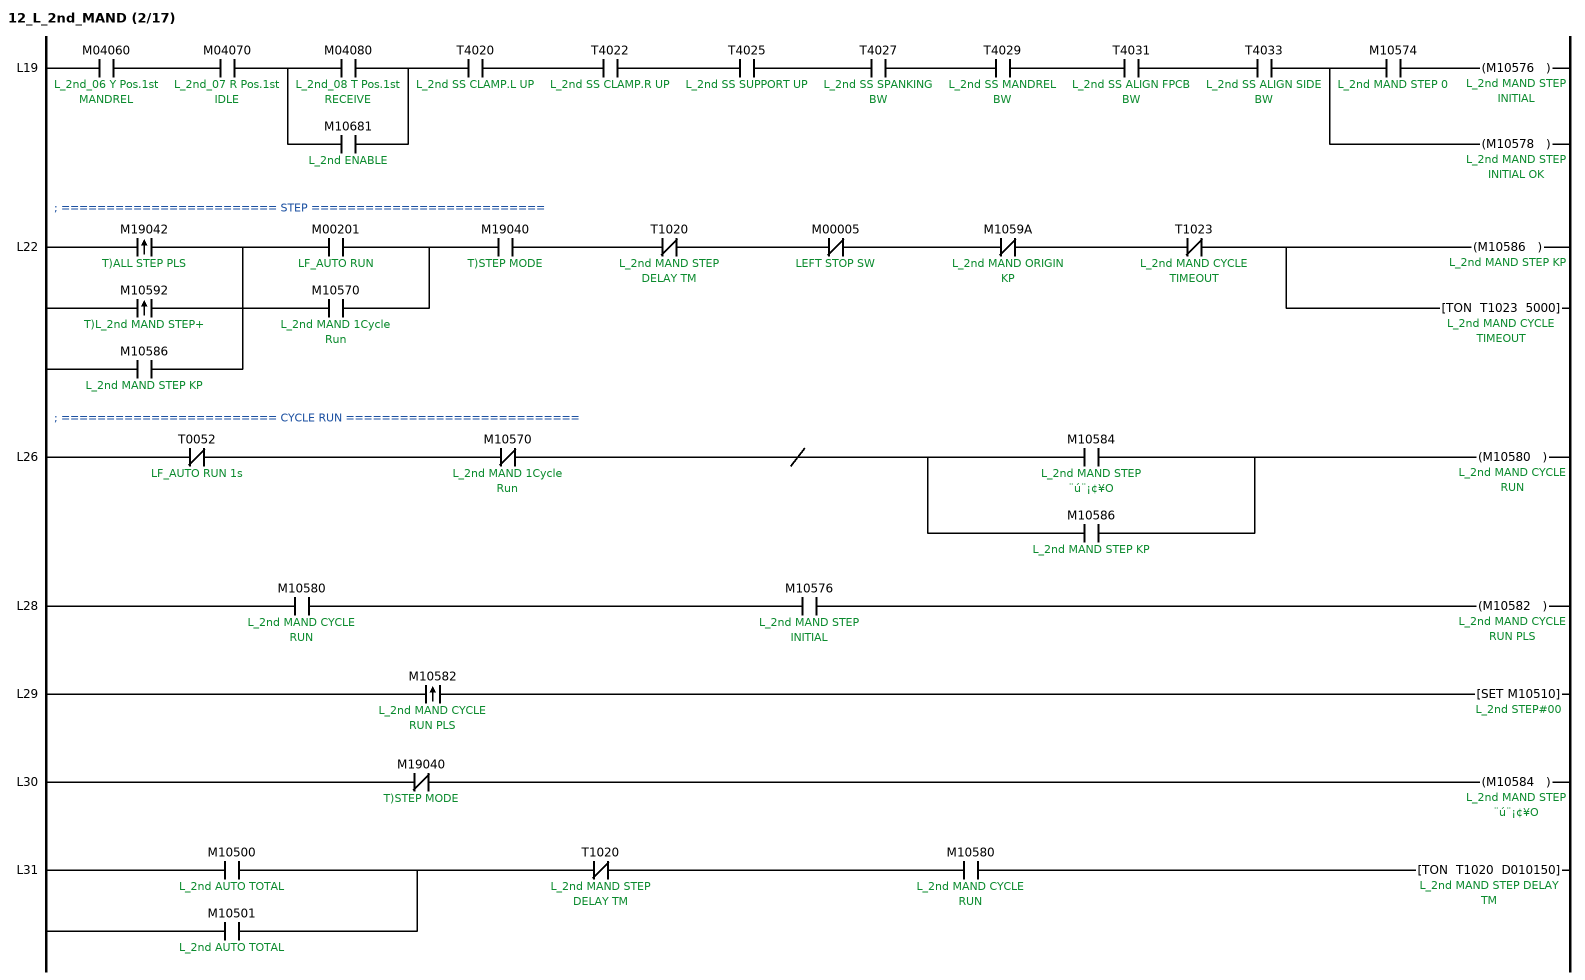
[picture p72: 12_L_2nd_MAND rungs L19-L31]
; L19
LOAD      M04060	// L_2nd_06 Y Pos.1st MANDREL
AND       M04070	// L_2nd_07 R Pos.1st IDLE
LOAD      M04080	// L_2nd_08 T Pos.1st RECEIVE
OR        M10681	// L_2nd ENABLE
AND LOAD
AND       T4020	// L_2nd SS CLAMP.L UP
AND       T4022	// L_2nd SS CLAMP.R UP
AND       T4025	// L_2nd SS SUPPORT UP
AND       T4027	// L_2nd SS SPANKING BW
AND       T4029	// L_2nd SS MANDREL BW
AND       T4031	// L_2nd SS ALIGN FPCB BW
AND       T4033	// L_2nd SS ALIGN SIDE BW
MPUSH
AND       M10574	// L_2nd MAND STEP 0
OUT       M10576	// L_2nd MAND STEP INITIAL
MPOP
OUT       M10578	// L_2nd MAND STEP INITIAL OK
// ======================== STEP ==========================
; L22
LOADP     M19042	// T)ALL STEP PLS
ORP       M10592	// T)L_2nd MAND STEP+
OR        M10586	// L_2nd MAND STEP KP
LOAD      M00201	// LF_AUTO RUN
OR        M10570	// L_2nd MAND 1Cycle Run
AND LOAD
AND       M19040	// T)STEP MODE
AND NOT   T1020	// L_2nd MAND STEP DELAY TM
AND NOT   M00005	// LEFT STOP SW
AND NOT   M1059A	// L_2nd MAND ORIGIN KP
AND NOT   T1023	// L_2nd MAND CYCLE TIMEOUT
OUT       M10586	// L_2nd MAND STEP KP
TON       T1023 5000	// L_2nd MAND CYCLE TIMEOUT
// ======================== CYCLE RUN ==========================
; L26
LOAD NOT  T0052	// LF_AUTO RUN 1s
AND NOT   M10570	// L_2nd MAND 1Cycle Run
NOT
LOAD      M10584	// L_2nd MAND STEP ¨ú¨¡¢¥O
OR        M10586	// L_2nd MAND STEP KP
AND LOAD
OUT       M10580	// L_2nd MAND CYCLE RUN
; L28
LOAD      M10580	// L_2nd MAND CYCLE RUN
AND       M10576	// L_2nd MAND STEP INITIAL
OUT       M10582	// L_2nd MAND CYCLE RUN PLS
; L29
LOADP     M10582	// L_2nd MAND CYCLE RUN PLS
SET       M10510	// L_2nd STEP#00
; L30
LOAD NOT  M19040	// T)STEP MODE
OUT       M10584	// L_2nd MAND STEP ¨ú¨¡¢¥O
; L31
LOAD      M10500	// L_2nd AUTO TOTAL
OR        M10501	// L_2nd AUTO TOTAL
AND NOT   T1020	// L_2nd MAND STEP DELAY TM
AND       M10580	// L_2nd MAND CYCLE RUN
TON       T1020 D010150	// L_2nd MAND STEP DELAY TM

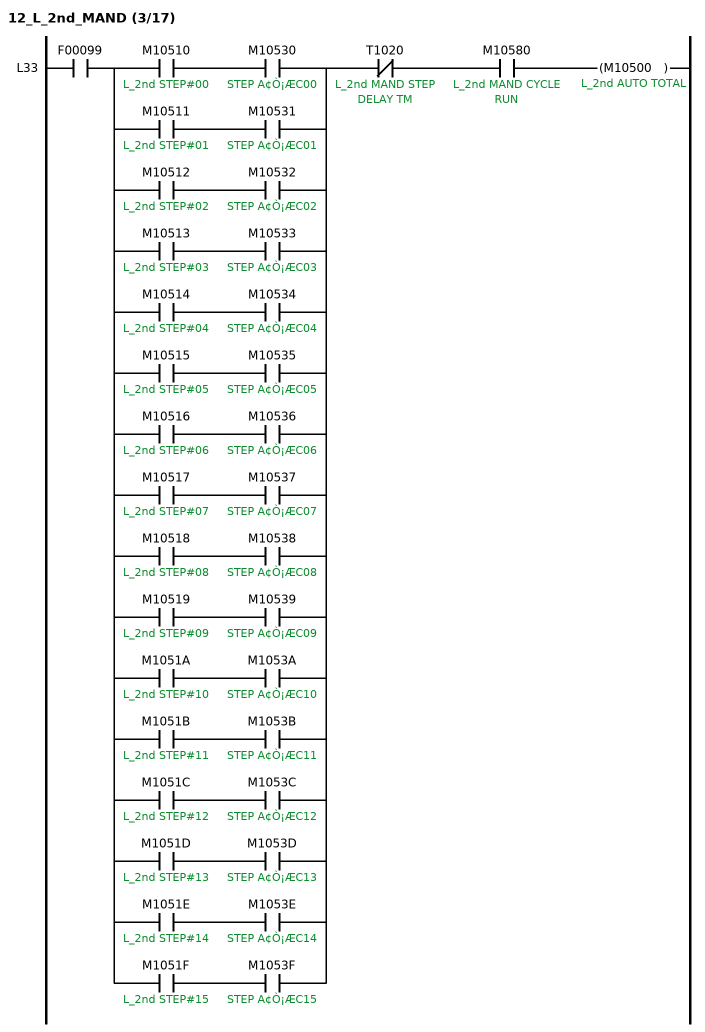
; L33
LOAD      F00099
LOAD      M10510	// L_2nd STEP#00
AND       M10530	// STEP A¢Ò¡ÆC00
LOAD      M10511	// L_2nd STEP#01
AND       M10531	// STEP A¢Ò¡ÆC01
OR LOAD
LOAD      M10512	// L_2nd STEP#02
AND       M10532	// STEP A¢Ò¡ÆC02
OR LOAD
LOAD      M10513	// L_2nd STEP#03
AND       M10533	// STEP A¢Ò¡ÆC03
OR LOAD
LOAD      M10514	// L_2nd STEP#04
AND       M10534	// STEP A¢Ò¡ÆC04
OR LOAD
LOAD      M10515	// L_2nd STEP#05
AND       M10535	// STEP A¢Ò¡ÆC05
OR LOAD
LOAD      M10516	// L_2nd STEP#06
AND       M10536	// STEP A¢Ò¡ÆC06
OR LOAD
LOAD      M10517	// L_2nd STEP#07
AND       M10537	// STEP A¢Ò¡ÆC07
OR LOAD
LOAD      M10518	// L_2nd STEP#08
AND       M10538	// STEP A¢Ò¡ÆC08
OR LOAD
LOAD      M10519	// L_2nd STEP#09
AND       M10539	// STEP A¢Ò¡ÆC09
OR LOAD
LOAD      M1051A	// L_2nd STEP#10
AND       M1053A	// STEP A¢Ò¡ÆC10
OR LOAD
LOAD      M1051B	// L_2nd STEP#11
AND       M1053B	// STEP A¢Ò¡ÆC11
OR LOAD
LOAD      M1051C	// L_2nd STEP#12
AND       M1053C	// STEP A¢Ò¡ÆC12
OR LOAD
LOAD      M1051D	// L_2nd STEP#13
AND       M1053D	// STEP A¢Ò¡ÆC13
OR LOAD
LOAD      M1051E	// L_2nd STEP#14
AND       M1053E	// STEP A¢Ò¡ÆC14
OR LOAD
LOAD      M1051F	// L_2nd STEP#15
AND       M1053F	// STEP A¢Ò¡ÆC15
OR LOAD
AND LOAD
AND NOT   T1020	// L_2nd MAND STEP DELAY TM
AND       M10580	// L_2nd MAND CYCLE RUN
OUT       M10500	// L_2nd AUTO TOTAL

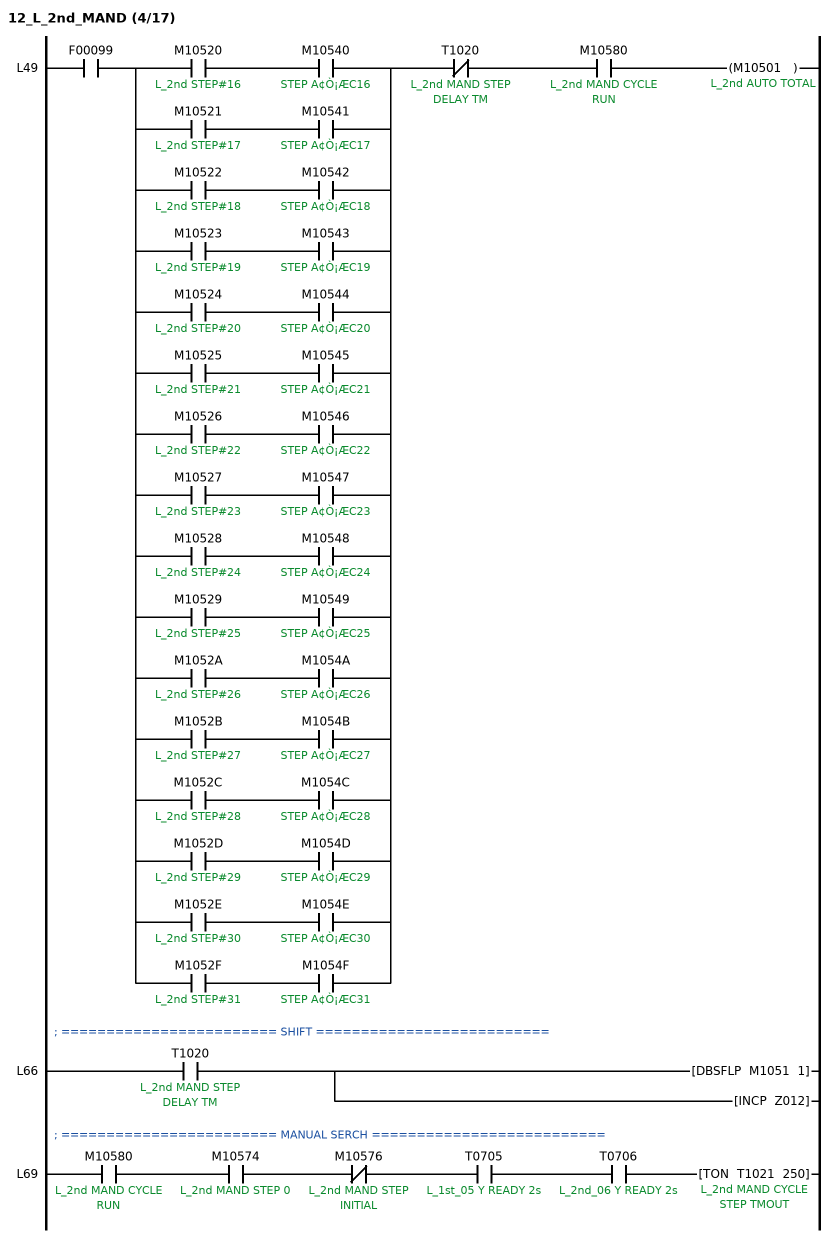
; L49
LOAD      F00099
LOAD      M10520	// L_2nd STEP#16
AND       M10540	// STEP A¢Ò¡ÆC16
LOAD      M10521	// L_2nd STEP#17
AND       M10541	// STEP A¢Ò¡ÆC17
OR LOAD
LOAD      M10522	// L_2nd STEP#18
AND       M10542	// STEP A¢Ò¡ÆC18
OR LOAD
LOAD      M10523	// L_2nd STEP#19
AND       M10543	// STEP A¢Ò¡ÆC19
OR LOAD
LOAD      M10524	// L_2nd STEP#20
AND       M10544	// STEP A¢Ò¡ÆC20
OR LOAD
LOAD      M10525	// L_2nd STEP#21
AND       M10545	// STEP A¢Ò¡ÆC21
OR LOAD
LOAD      M10526	// L_2nd STEP#22
AND       M10546	// STEP A¢Ò¡ÆC22
OR LOAD
LOAD      M10527	// L_2nd STEP#23
AND       M10547	// STEP A¢Ò¡ÆC23
OR LOAD
LOAD      M10528	// L_2nd STEP#24
AND       M10548	// STEP A¢Ò¡ÆC24
OR LOAD
LOAD      M10529	// L_2nd STEP#25
AND       M10549	// STEP A¢Ò¡ÆC25
OR LOAD
LOAD      M1052A	// L_2nd STEP#26
AND       M1054A	// STEP A¢Ò¡ÆC26
OR LOAD
LOAD      M1052B	// L_2nd STEP#27
AND       M1054B	// STEP A¢Ò¡ÆC27
OR LOAD
LOAD      M1052C	// L_2nd STEP#28
AND       M1054C	// STEP A¢Ò¡ÆC28
OR LOAD
LOAD      M1052D	// L_2nd STEP#29
AND       M1054D	// STEP A¢Ò¡ÆC29
OR LOAD
LOAD      M1052E	// L_2nd STEP#30
AND       M1054E	// STEP A¢Ò¡ÆC30
OR LOAD
LOAD      M1052F	// L_2nd STEP#31
AND       M1054F	// STEP A¢Ò¡ÆC31
OR LOAD
AND LOAD
AND NOT   T1020	// L_2nd MAND STEP DELAY TM
AND       M10580	// L_2nd MAND CYCLE RUN
OUT       M10501	// L_2nd AUTO TOTAL
// ======================== SHIFT ==========================
; L66
LOAD      T1020	// L_2nd MAND STEP DELAY TM
DBSFLP    M1051 1
INCP      Z012
// ======================== MANUAL SERCH ==========================
; L69
LOAD      M10580	// L_2nd MAND CYCLE RUN
AND       M10574	// L_2nd MAND STEP 0
AND NOT   M10576	// L_2nd MAND STEP INITIAL
AND       T0705	// L_1st_05 Y READY 2s
AND       T0706	// L_2nd_06 Y READY 2s
TON       T1021 250	// L_2nd MAND CYCLE STEP TMOUT

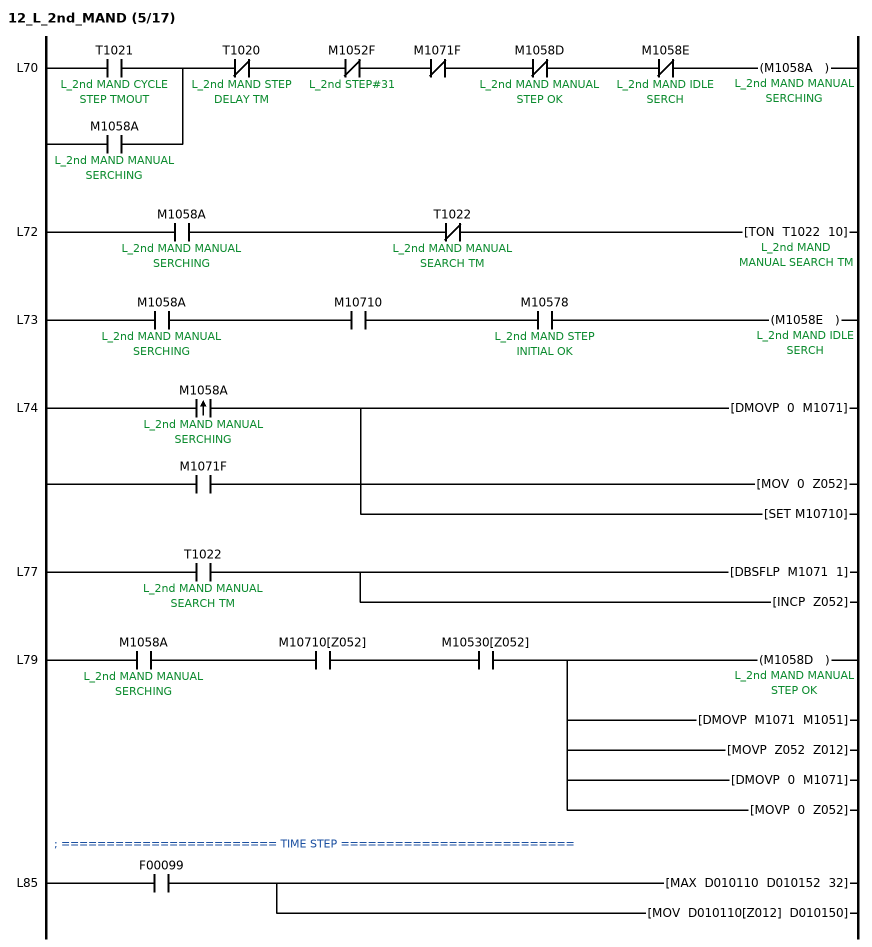
; L70
LOAD      T1021	// L_2nd MAND CYCLE STEP TMOUT
OR        M1058A	// L_2nd MAND MANUAL SERCHING
AND NOT   T1020	// L_2nd MAND STEP DELAY TM
AND NOT   M1052F	// L_2nd STEP#31
AND NOT   M1071F
AND NOT   M1058D	// L_2nd MAND MANUAL STEP OK
AND NOT   M1058E	// L_2nd MAND IDLE SERCH
OUT       M1058A	// L_2nd MAND MANUAL SERCHING
; L72
LOAD      M1058A	// L_2nd MAND MANUAL SERCHING
AND NOT   T1022	// L_2nd MAND MANUAL SEARCH TM
TON       T1022 10	// L_2nd MAND MANUAL SEARCH TM
; L73
LOAD      M1058A	// L_2nd MAND MANUAL SERCHING
AND       M10710
AND       M10578	// L_2nd MAND STEP INITIAL OK
OUT       M1058E	// L_2nd MAND IDLE SERCH
; L74
LOADP     M1058A	// L_2nd MAND MANUAL SERCHING
OR        M1071F
DMOVP     0 M1071
MOV       0 Z052
SET       M10710
; L77
LOAD      T1022	// L_2nd MAND MANUAL SEARCH TM
DBSFLP    M1071 1
INCP      Z052
; L79
LOAD      M1058A	// L_2nd MAND MANUAL SERCHING
AND       M10710[Z052]
AND       M10530[Z052]
OUT       M1058D	// L_2nd MAND MANUAL STEP OK
DMOVP     M1071 M1051
MOVP      Z052 Z012
DMOVP     0 M1071
MOVP      0 Z052
// ======================== TIME STEP ==========================
; L85
LOAD      F00099
MAX       D010110 D010152 32
MOV       D010110[Z012] D010150

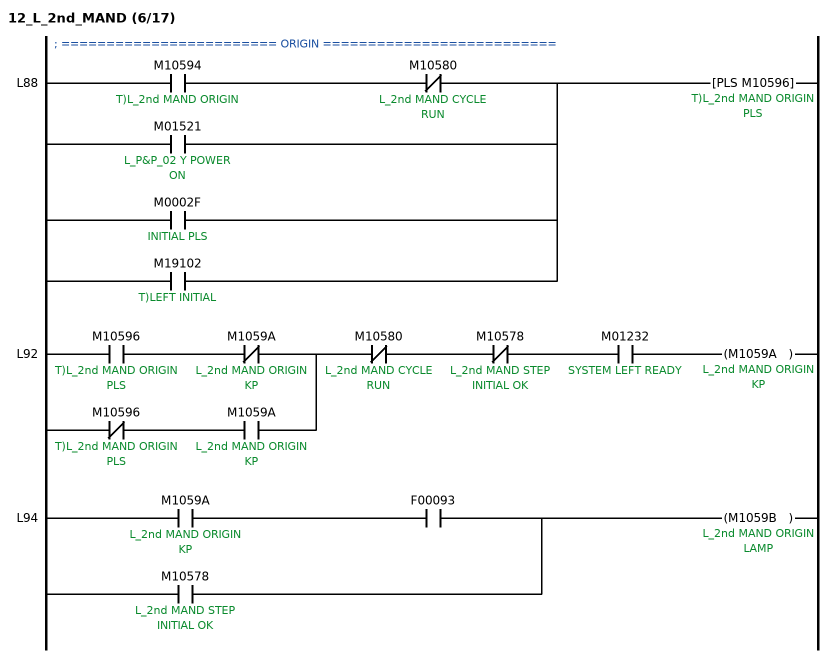
// ======================== ORIGIN ==========================
; L88
LOAD      M10594	// T)L_2nd MAND ORIGIN
AND NOT   M10580	// L_2nd MAND CYCLE RUN
OR        M01521	// L_P&P_02 Y POWER ON
OR        M0002F	// INITIAL PLS
OR        M19102	// T)LEFT INITIAL
OUTP      M10596	// T)L_2nd MAND ORIGIN PLS
; L92
LOAD      M10596	// T)L_2nd MAND ORIGIN PLS
AND NOT   M1059A	// L_2nd MAND ORIGIN KP
LOAD NOT  M10596	// T)L_2nd MAND ORIGIN PLS
AND       M1059A	// L_2nd MAND ORIGIN KP
OR LOAD
AND NOT   M10580	// L_2nd MAND CYCLE RUN
AND NOT   M10578	// L_2nd MAND STEP INITIAL OK
AND       M01232	// SYSTEM LEFT READY
OUT       M1059A	// L_2nd MAND ORIGIN KP
; L94
LOAD      M1059A	// L_2nd MAND ORIGIN KP
AND       F00093
OR        M10578	// L_2nd MAND STEP INITIAL OK
OUT       M1059B	// L_2nd MAND ORIGIN LAMP

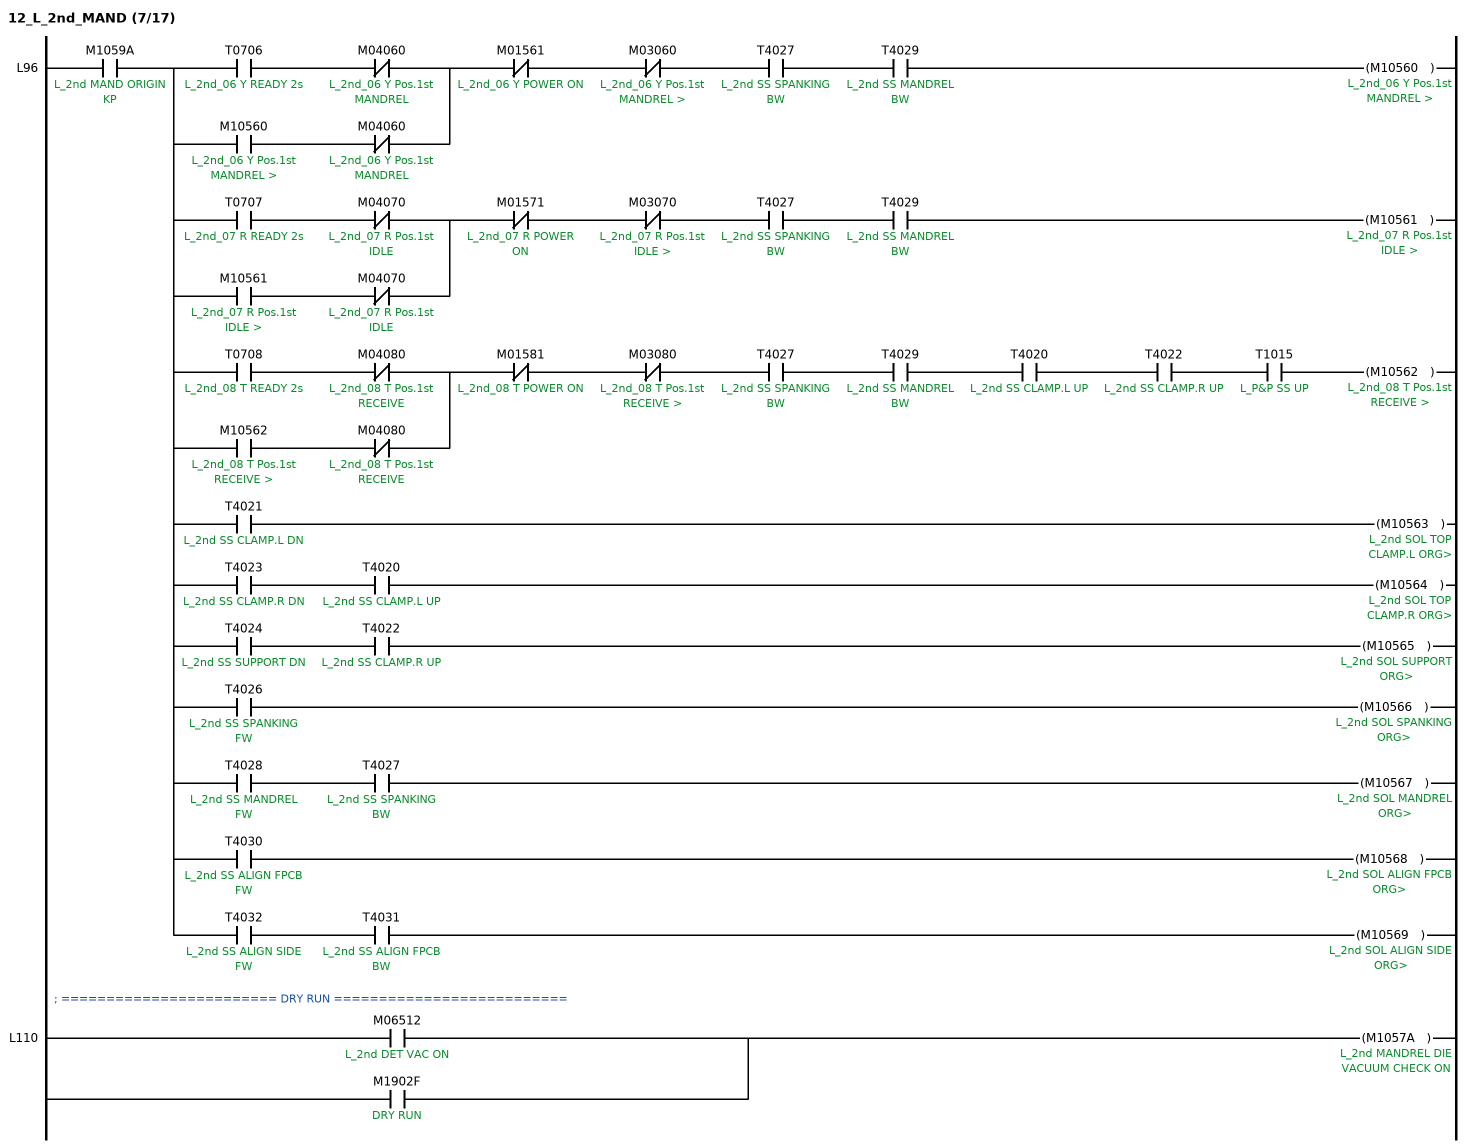
; L96
LOAD      M1059A	// L_2nd MAND ORIGIN KP
MPUSH
LOAD      T0706	// L_2nd_06 Y READY 2s
AND NOT   M04060	// L_2nd_06 Y Pos.1st MANDREL
LOAD      M10560	// L_2nd_06 Y Pos.1st MANDREL >
AND NOT   M04060	// L_2nd_06 Y Pos.1st MANDREL
OR LOAD
AND LOAD
AND NOT   M01561	// L_2nd_06 Y POWER ON
AND NOT   M03060	// L_2nd_06 Y Pos.1st MANDREL >
AND       T4027	// L_2nd SS SPANKING BW
AND       T4029	// L_2nd SS MANDREL BW
OUT       M10560	// L_2nd_06 Y Pos.1st MANDREL >
MLOAD
LOAD      T0707	// L_2nd_07 R READY 2s
AND NOT   M04070	// L_2nd_07 R Pos.1st IDLE
LOAD      M10561	// L_2nd_07 R Pos.1st IDLE >
AND NOT   M04070	// L_2nd_07 R Pos.1st IDLE
OR LOAD
AND LOAD
AND NOT   M01571	// L_2nd_07 R POWER ON
AND NOT   M03070	// L_2nd_07 R Pos.1st IDLE >
AND       T4027	// L_2nd SS SPANKING BW
AND       T4029	// L_2nd SS MANDREL BW
OUT       M10561	// L_2nd_07 R Pos.1st IDLE >
MLOAD
LOAD      T0708	// L_2nd_08 T READY 2s
AND NOT   M04080	// L_2nd_08 T Pos.1st RECEIVE
LOAD      M10562	// L_2nd_08 T Pos.1st RECEIVE >
AND NOT   M04080	// L_2nd_08 T Pos.1st RECEIVE
OR LOAD
AND LOAD
AND NOT   M01581	// L_2nd_08 T POWER ON
AND NOT   M03080	// L_2nd_08 T Pos.1st RECEIVE >
AND       T4027	// L_2nd SS SPANKING BW
AND       T4029	// L_2nd SS MANDREL BW
AND       T4020	// L_2nd SS CLAMP.L UP
AND       T4022	// L_2nd SS CLAMP.R UP
AND       T1015	// L_P&P SS UP
OUT       M10562	// L_2nd_08 T Pos.1st RECEIVE >
MLOAD
AND       T4021	// L_2nd SS CLAMP.L DN
OUT       M10563	// L_2nd SOL TOP CLAMP.L ORG>
MLOAD
AND       T4023	// L_2nd SS CLAMP.R DN
AND       T4020	// L_2nd SS CLAMP.L UP
OUT       M10564	// L_2nd SOL TOP CLAMP.R ORG>
MLOAD
AND       T4024	// L_2nd SS SUPPORT DN
AND       T4022	// L_2nd SS CLAMP.R UP
OUT       M10565	// L_2nd SOL SUPPORT ORG>
MLOAD
AND       T4026	// L_2nd SS SPANKING FW
OUT       M10566	// L_2nd SOL SPANKING ORG>
MLOAD
AND       T4028	// L_2nd SS MANDREL FW
AND       T4027	// L_2nd SS SPANKING BW
OUT       M10567	// L_2nd SOL MANDREL ORG>
MLOAD
AND       T4030	// L_2nd SS ALIGN FPCB FW
OUT       M10568	// L_2nd SOL ALIGN FPCB ORG>
MPOP
AND       T4032	// L_2nd SS ALIGN SIDE FW
AND       T4031	// L_2nd SS ALIGN FPCB BW
OUT       M10569	// L_2nd SOL ALIGN SIDE ORG>
// ======================== DRY RUN ==========================
; L110
LOAD      M06512	// L_2nd DET VAC ON
OR        M1902F	// DRY RUN
OUT       M1057A	// L_2nd MANDREL DIE VACUUM CHECK ON

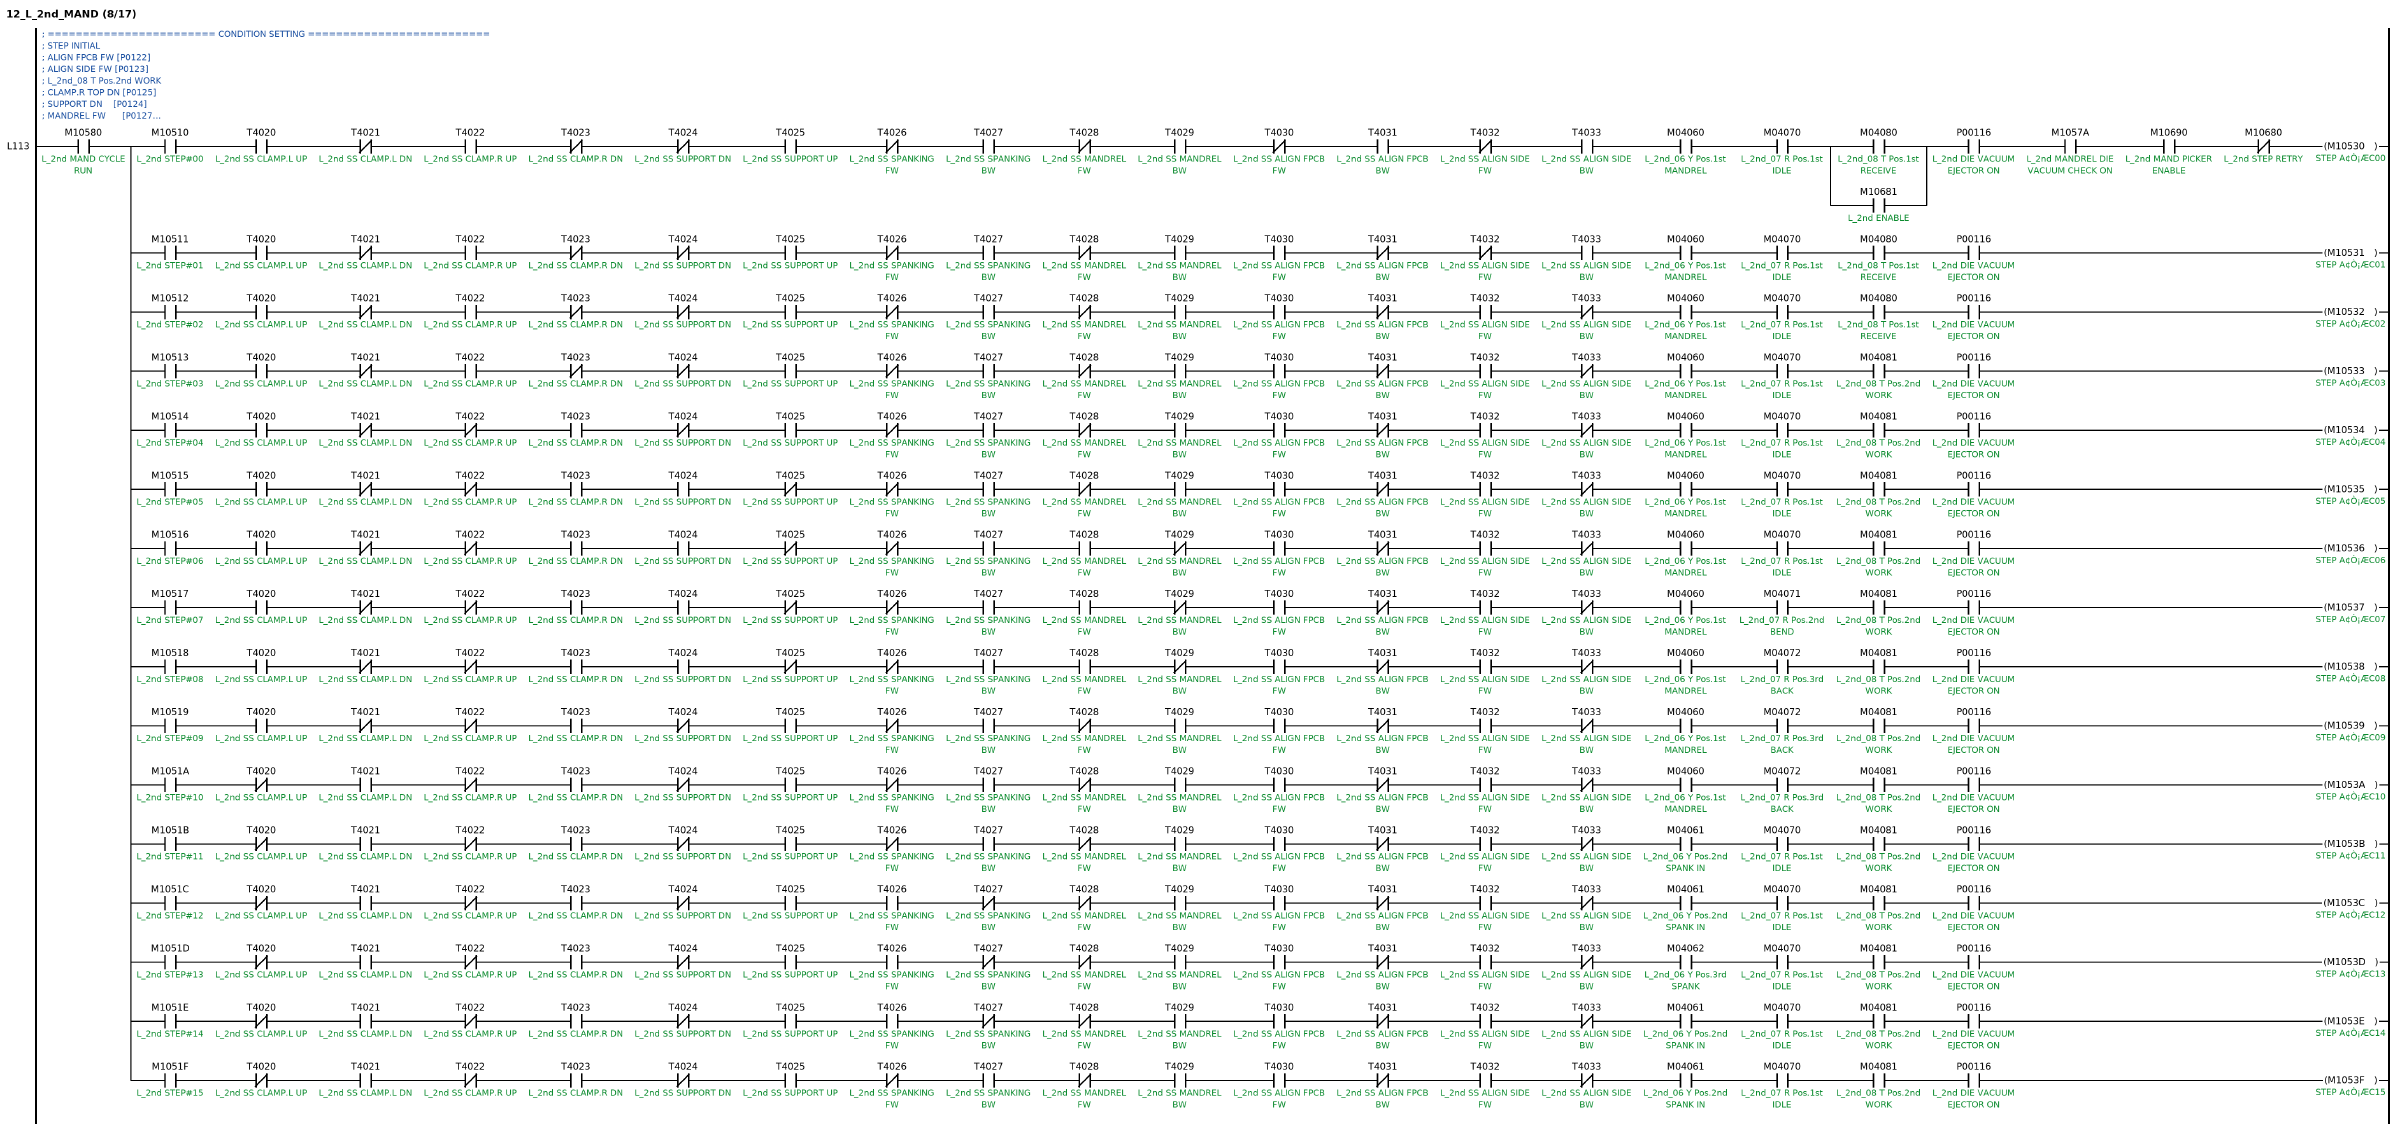
// ======================== CONDITION SETTING ==========================
; L113
LOAD      M10580	// L_2nd MAND CYCLE RUN
MPUSH
AND       M10510	// L_2nd STEP#00
AND       T4020	// L_2nd SS CLAMP.L UP
AND NOT   T4021	// L_2nd SS CLAMP.L DN
AND       T4022	// L_2nd SS CLAMP.R UP
AND NOT   T4023	// L_2nd SS CLAMP.R DN
AND NOT   T4024	// L_2nd SS SUPPORT DN
AND       T4025	// L_2nd SS SUPPORT UP
AND NOT   T4026	// L_2nd SS SPANKING FW
AND       T4027	// L_2nd SS SPANKING BW
AND NOT   T4028	// L_2nd SS MANDREL FW
AND       T4029	// L_2nd SS MANDREL BW
AND NOT   T4030	// L_2nd SS ALIGN FPCB FW
AND       T4031	// L_2nd SS ALIGN FPCB BW
AND NOT   T4032	// L_2nd SS ALIGN SIDE FW
AND       T4033	// L_2nd SS ALIGN SIDE BW
AND       M04060	// L_2nd_06 Y Pos.1st MANDREL
AND       M04070	// L_2nd_07 R Pos.1st IDLE
LOAD      M04080	// L_2nd_08 T Pos.1st RECEIVE
OR        M10681	// L_2nd ENABLE
AND LOAD
AND       P00116	// L_2nd DIE VACUUM EJECTOR ON
AND       M1057A	// L_2nd MANDREL DIE VACUUM CHECK ON
AND       M10690	// L_2nd MAND PICKER ENABLE
AND NOT   M10680	// L_2nd STEP RETRY
OUT       M10530	// STEP A¢Ò¡ÆC00
MLOAD
AND       M10511	// L_2nd STEP#01
AND       T4020	// L_2nd SS CLAMP.L UP
AND NOT   T4021	// L_2nd SS CLAMP.L DN
AND       T4022	// L_2nd SS CLAMP.R UP
AND NOT   T4023	// L_2nd SS CLAMP.R DN
AND NOT   T4024	// L_2nd SS SUPPORT DN
AND       T4025	// L_2nd SS SUPPORT UP
AND NOT   T4026	// L_2nd SS SPANKING FW
AND       T4027	// L_2nd SS SPANKING BW
AND NOT   T4028	// L_2nd SS MANDREL FW
AND       T4029	// L_2nd SS MANDREL BW
AND       T4030	// L_2nd SS ALIGN FPCB FW
AND NOT   T4031	// L_2nd SS ALIGN FPCB BW
AND NOT   T4032	// L_2nd SS ALIGN SIDE FW
AND       T4033	// L_2nd SS ALIGN SIDE BW
AND       M04060	// L_2nd_06 Y Pos.1st MANDREL
AND       M04070	// L_2nd_07 R Pos.1st IDLE
AND       M04080	// L_2nd_08 T Pos.1st RECEIVE
AND       P00116	// L_2nd DIE VACUUM EJECTOR ON
OUT       M10531	// STEP A¢Ò¡ÆC01
MLOAD
AND       M10512	// L_2nd STEP#02
AND       T4020	// L_2nd SS CLAMP.L UP
AND NOT   T4021	// L_2nd SS CLAMP.L DN
AND       T4022	// L_2nd SS CLAMP.R UP
AND NOT   T4023	// L_2nd SS CLAMP.R DN
AND NOT   T4024	// L_2nd SS SUPPORT DN
AND       T4025	// L_2nd SS SUPPORT UP
AND NOT   T4026	// L_2nd SS SPANKING FW
AND       T4027	// L_2nd SS SPANKING BW
AND NOT   T4028	// L_2nd SS MANDREL FW
AND       T4029	// L_2nd SS MANDREL BW
AND       T4030	// L_2nd SS ALIGN FPCB FW
AND NOT   T4031	// L_2nd SS ALIGN FPCB BW
AND       T4032	// L_2nd SS ALIGN SIDE FW
AND NOT   T4033	// L_2nd SS ALIGN SIDE BW
AND       M04060	// L_2nd_06 Y Pos.1st MANDREL
AND       M04070	// L_2nd_07 R Pos.1st IDLE
AND       M04080	// L_2nd_08 T Pos.1st RECEIVE
AND       P00116	// L_2nd DIE VACUUM EJECTOR ON
OUT       M10532	// STEP A¢Ò¡ÆC02
MLOAD
AND       M10513	// L_2nd STEP#03
AND       T4020	// L_2nd SS CLAMP.L UP
AND NOT   T4021	// L_2nd SS CLAMP.L DN
AND       T4022	// L_2nd SS CLAMP.R UP
AND NOT   T4023	// L_2nd SS CLAMP.R DN
AND NOT   T4024	// L_2nd SS SUPPORT DN
AND       T4025	// L_2nd SS SUPPORT UP
AND NOT   T4026	// L_2nd SS SPANKING FW
AND       T4027	// L_2nd SS SPANKING BW
AND NOT   T4028	// L_2nd SS MANDREL FW
AND       T4029	// L_2nd SS MANDREL BW
AND       T4030	// L_2nd SS ALIGN FPCB FW
AND NOT   T4031	// L_2nd SS ALIGN FPCB BW
AND       T4032	// L_2nd SS ALIGN SIDE FW
AND NOT   T4033	// L_2nd SS ALIGN SIDE BW
AND       M04060	// L_2nd_06 Y Pos.1st MANDREL
AND       M04070	// L_2nd_07 R Pos.1st IDLE
AND       M04081	// L_2nd_08 T Pos.2nd WORK
AND       P00116	// L_2nd DIE VACUUM EJECTOR ON
OUT       M10533	// STEP A¢Ò¡ÆC03
MLOAD
AND       M10514	// L_2nd STEP#04
AND       T4020	// L_2nd SS CLAMP.L UP
AND NOT   T4021	// L_2nd SS CLAMP.L DN
AND NOT   T4022	// L_2nd SS CLAMP.R UP
AND       T4023	// L_2nd SS CLAMP.R DN
AND NOT   T4024	// L_2nd SS SUPPORT DN
AND       T4025	// L_2nd SS SUPPORT UP
AND NOT   T4026	// L_2nd SS SPANKING FW
AND       T4027	// L_2nd SS SPANKING BW
AND NOT   T4028	// L_2nd SS MANDREL FW
AND       T4029	// L_2nd SS MANDREL BW
AND       T4030	// L_2nd SS ALIGN FPCB FW
AND NOT   T4031	// L_2nd SS ALIGN FPCB BW
AND       T4032	// L_2nd SS ALIGN SIDE FW
AND NOT   T4033	// L_2nd SS ALIGN SIDE BW
AND       M04060	// L_2nd_06 Y Pos.1st MANDREL
AND       M04070	// L_2nd_07 R Pos.1st IDLE
AND       M04081	// L_2nd_08 T Pos.2nd WORK
AND       P00116	// L_2nd DIE VACUUM EJECTOR ON
OUT       M10534	// STEP A¢Ò¡ÆC04
MLOAD
AND       M10515	// L_2nd STEP#05
AND       T4020	// L_2nd SS CLAMP.L UP
AND NOT   T4021	// L_2nd SS CLAMP.L DN
AND NOT   T4022	// L_2nd SS CLAMP.R UP
AND       T4023	// L_2nd SS CLAMP.R DN
AND       T4024	// L_2nd SS SUPPORT DN
AND NOT   T4025	// L_2nd SS SUPPORT UP
AND NOT   T4026	// L_2nd SS SPANKING FW
AND       T4027	// L_2nd SS SPANKING BW
AND NOT   T4028	// L_2nd SS MANDREL FW
AND       T4029	// L_2nd SS MANDREL BW
AND       T4030	// L_2nd SS ALIGN FPCB FW
AND NOT   T4031	// L_2nd SS ALIGN FPCB BW
AND       T4032	// L_2nd SS ALIGN SIDE FW
AND NOT   T4033	// L_2nd SS ALIGN SIDE BW
AND       M04060	// L_2nd_06 Y Pos.1st MANDREL
AND       M04070	// L_2nd_07 R Pos.1st IDLE
AND       M04081	// L_2nd_08 T Pos.2nd WORK
AND       P00116	// L_2nd DIE VACUUM EJECTOR ON
OUT       M10535	// STEP A¢Ò¡ÆC05
MLOAD
AND       M10516	// L_2nd STEP#06
AND       T4020	// L_2nd SS CLAMP.L UP
AND NOT   T4021	// L_2nd SS CLAMP.L DN
AND NOT   T4022	// L_2nd SS CLAMP.R UP
AND       T4023	// L_2nd SS CLAMP.R DN
AND       T4024	// L_2nd SS SUPPORT DN
AND NOT   T4025	// L_2nd SS SUPPORT UP
AND NOT   T4026	// L_2nd SS SPANKING FW
AND       T4027	// L_2nd SS SPANKING BW
AND       T4028	// L_2nd SS MANDREL FW
AND NOT   T4029	// L_2nd SS MANDREL BW
AND       T4030	// L_2nd SS ALIGN FPCB FW
AND NOT   T4031	// L_2nd SS ALIGN FPCB BW
AND       T4032	// L_2nd SS ALIGN SIDE FW
AND NOT   T4033	// L_2nd SS ALIGN SIDE BW
AND       M04060	// L_2nd_06 Y Pos.1st MANDREL
AND       M04070	// L_2nd_07 R Pos.1st IDLE
AND       M04081	// L_2nd_08 T Pos.2nd WORK
AND       P00116	// L_2nd DIE VACUUM EJECTOR ON
OUT       M10536	// STEP A¢Ò¡ÆC06
MLOAD
AND       M10517	// L_2nd STEP#07
AND       T4020	// L_2nd SS CLAMP.L UP
AND NOT   T4021	// L_2nd SS CLAMP.L DN
AND NOT   T4022	// L_2nd SS CLAMP.R UP
AND       T4023	// L_2nd SS CLAMP.R DN
AND       T4024	// L_2nd SS SUPPORT DN
AND NOT   T4025	// L_2nd SS SUPPORT UP
AND NOT   T4026	// L_2nd SS SPANKING FW
AND       T4027	// L_2nd SS SPANKING BW
AND       T4028	// L_2nd SS MANDREL FW
AND NOT   T4029	// L_2nd SS MANDREL BW
AND       T4030	// L_2nd SS ALIGN FPCB FW
AND NOT   T4031	// L_2nd SS ALIGN FPCB BW
AND       T4032	// L_2nd SS ALIGN SIDE FW
AND NOT   T4033	// L_2nd SS ALIGN SIDE BW
AND       M04060	// L_2nd_06 Y Pos.1st MANDREL
AND       M04071	// L_2nd_07 R Pos.2nd BEND
AND       M04081	// L_2nd_08 T Pos.2nd WORK
AND       P00116	// L_2nd DIE VACUUM EJECTOR ON
OUT       M10537	// STEP A¢Ò¡ÆC07
MLOAD
AND       M10518	// L_2nd STEP#08
AND       T4020	// L_2nd SS CLAMP.L UP
AND NOT   T4021	// L_2nd SS CLAMP.L DN
AND NOT   T4022	// L_2nd SS CLAMP.R UP
AND       T4023	// L_2nd SS CLAMP.R DN
AND       T4024	// L_2nd SS SUPPORT DN
AND NOT   T4025	// L_2nd SS SUPPORT UP
AND NOT   T4026	// L_2nd SS SPANKING FW
AND       T4027	// L_2nd SS SPANKING BW
AND       T4028	// L_2nd SS MANDREL FW
AND NOT   T4029	// L_2nd SS MANDREL BW
AND       T4030	// L_2nd SS ALIGN FPCB FW
AND NOT   T4031	// L_2nd SS ALIGN FPCB BW
AND       T4032	// L_2nd SS ALIGN SIDE FW
AND NOT   T4033	// L_2nd SS ALIGN SIDE BW
AND       M04060	// L_2nd_06 Y Pos.1st MANDREL
AND       M04072	// L_2nd_07 R Pos.3rd BACK
AND       M04081	// L_2nd_08 T Pos.2nd WORK
AND       P00116	// L_2nd DIE VACUUM EJECTOR ON
OUT       M10538	// STEP A¢Ò¡ÆC08
MLOAD
AND       M10519	// L_2nd STEP#09
AND       T4020	// L_2nd SS CLAMP.L UP
AND NOT   T4021	// L_2nd SS CLAMP.L DN
AND NOT   T4022	// L_2nd SS CLAMP.R UP
AND       T4023	// L_2nd SS CLAMP.R DN
AND NOT   T4024	// L_2nd SS SUPPORT DN
AND       T4025	// L_2nd SS SUPPORT UP
AND NOT   T4026	// L_2nd SS SPANKING FW
AND       T4027	// L_2nd SS SPANKING BW
AND NOT   T4028	// L_2nd SS MANDREL FW
AND       T4029	// L_2nd SS MANDREL BW
AND       T4030	// L_2nd SS ALIGN FPCB FW
AND NOT   T4031	// L_2nd SS ALIGN FPCB BW
AND       T4032	// L_2nd SS ALIGN SIDE FW
AND NOT   T4033	// L_2nd SS ALIGN SIDE BW
AND       M04060	// L_2nd_06 Y Pos.1st MANDREL
AND       M04072	// L_2nd_07 R Pos.3rd BACK
AND       M04081	// L_2nd_08 T Pos.2nd WORK
AND       P00116	// L_2nd DIE VACUUM EJECTOR ON
OUT       M10539	// STEP A¢Ò¡ÆC09
MLOAD
AND       M1051A	// L_2nd STEP#10
AND NOT   T4020	// L_2nd SS CLAMP.L UP
AND       T4021	// L_2nd SS CLAMP.L DN
AND NOT   T4022	// L_2nd SS CLAMP.R UP
AND       T4023	// L_2nd SS CLAMP.R DN
AND NOT   T4024	// L_2nd SS SUPPORT DN
AND       T4025	// L_2nd SS SUPPORT UP
AND NOT   T4026	// L_2nd SS SPANKING FW
AND       T4027	// L_2nd SS SPANKING BW
AND NOT   T4028	// L_2nd SS MANDREL FW
AND       T4029	// L_2nd SS MANDREL BW
AND       T4030	// L_2nd SS ALIGN FPCB FW
AND NOT   T4031	// L_2nd SS ALIGN FPCB BW
AND       T4032	// L_2nd SS ALIGN SIDE FW
AND NOT   T4033	// L_2nd SS ALIGN SIDE BW
AND       M04060	// L_2nd_06 Y Pos.1st MANDREL
AND       M04072	// L_2nd_07 R Pos.3rd BACK
AND       M04081	// L_2nd_08 T Pos.2nd WORK
AND       P00116	// L_2nd DIE VACUUM EJECTOR ON
OUT       M1053A	// STEP A¢Ò¡ÆC10
MLOAD
AND       M1051B	// L_2nd STEP#11
AND NOT   T4020	// L_2nd SS CLAMP.L UP
AND       T4021	// L_2nd SS CLAMP.L DN
AND NOT   T4022	// L_2nd SS CLAMP.R UP
AND       T4023	// L_2nd SS CLAMP.R DN
AND NOT   T4024	// L_2nd SS SUPPORT DN
AND       T4025	// L_2nd SS SUPPORT UP
AND NOT   T4026	// L_2nd SS SPANKING FW
AND       T4027	// L_2nd SS SPANKING BW
AND NOT   T4028	// L_2nd SS MANDREL FW
AND       T4029	// L_2nd SS MANDREL BW
AND       T4030	// L_2nd SS ALIGN FPCB FW
AND NOT   T4031	// L_2nd SS ALIGN FPCB BW
AND       T4032	// L_2nd SS ALIGN SIDE FW
AND NOT   T4033	// L_2nd SS ALIGN SIDE BW
AND       M04061	// L_2nd_06 Y Pos.2nd SPANK IN
AND       M04070	// L_2nd_07 R Pos.1st IDLE
AND       M04081	// L_2nd_08 T Pos.2nd WORK
AND       P00116	// L_2nd DIE VACUUM EJECTOR ON
OUT       M1053B	// STEP A¢Ò¡ÆC11
MLOAD
AND       M1051C	// L_2nd STEP#12
AND NOT   T4020	// L_2nd SS CLAMP.L UP
AND       T4021	// L_2nd SS CLAMP.L DN
AND NOT   T4022	// L_2nd SS CLAMP.R UP
AND       T4023	// L_2nd SS CLAMP.R DN
AND NOT   T4024	// L_2nd SS SUPPORT DN
AND       T4025	// L_2nd SS SUPPORT UP
AND       T4026	// L_2nd SS SPANKING FW
AND NOT   T4027	// L_2nd SS SPANKING BW
AND NOT   T4028	// L_2nd SS MANDREL FW
AND       T4029	// L_2nd SS MANDREL BW
AND       T4030	// L_2nd SS ALIGN FPCB FW
AND NOT   T4031	// L_2nd SS ALIGN FPCB BW
AND       T4032	// L_2nd SS ALIGN SIDE FW
AND NOT   T4033	// L_2nd SS ALIGN SIDE BW
AND       M04061	// L_2nd_06 Y Pos.2nd SPANK IN
AND       M04070	// L_2nd_07 R Pos.1st IDLE
AND       M04081	// L_2nd_08 T Pos.2nd WORK
AND       P00116	// L_2nd DIE VACUUM EJECTOR ON
OUT       M1053C	// STEP A¢Ò¡ÆC12
MLOAD
AND       M1051D	// L_2nd STEP#13
AND NOT   T4020	// L_2nd SS CLAMP.L UP
AND       T4021	// L_2nd SS CLAMP.L DN
AND NOT   T4022	// L_2nd SS CLAMP.R UP
AND       T4023	// L_2nd SS CLAMP.R DN
AND NOT   T4024	// L_2nd SS SUPPORT DN
AND       T4025	// L_2nd SS SUPPORT UP
AND       T4026	// L_2nd SS SPANKING FW
AND NOT   T4027	// L_2nd SS SPANKING BW
AND NOT   T4028	// L_2nd SS MANDREL FW
AND       T4029	// L_2nd SS MANDREL BW
AND       T4030	// L_2nd SS ALIGN FPCB FW
AND NOT   T4031	// L_2nd SS ALIGN FPCB BW
AND       T4032	// L_2nd SS ALIGN SIDE FW
AND NOT   T4033	// L_2nd SS ALIGN SIDE BW
AND       M04062	// L_2nd_06 Y Pos.3rd SPANK
AND       M04070	// L_2nd_07 R Pos.1st IDLE
AND       M04081	// L_2nd_08 T Pos.2nd WORK
AND       P00116	// L_2nd DIE VACUUM EJECTOR ON
OUT       M1053D	// STEP A¢Ò¡ÆC13
MLOAD
AND       M1051E	// L_2nd STEP#14
AND NOT   T4020	// L_2nd SS CLAMP.L UP
AND       T4021	// L_2nd SS CLAMP.L DN
AND NOT   T4022	// L_2nd SS CLAMP.R UP
AND       T4023	// L_2nd SS CLAMP.R DN
AND NOT   T4024	// L_2nd SS SUPPORT DN
AND       T4025	// L_2nd SS SUPPORT UP
AND       T4026	// L_2nd SS SPANKING FW
AND NOT   T4027	// L_2nd SS SPANKING BW
AND NOT   T4028	// L_2nd SS MANDREL FW
AND       T4029	// L_2nd SS MANDREL BW
AND       T4030	// L_2nd SS ALIGN FPCB FW
AND NOT   T4031	// L_2nd SS ALIGN FPCB BW
AND       T4032	// L_2nd SS ALIGN SIDE FW
AND NOT   T4033	// L_2nd SS ALIGN SIDE BW
AND       M04061	// L_2nd_06 Y Pos.2nd SPANK IN
AND       M04070	// L_2nd_07 R Pos.1st IDLE
AND       M04081	// L_2nd_08 T Pos.2nd WORK
AND       P00116	// L_2nd DIE VACUUM EJECTOR ON
OUT       M1053E	// STEP A¢Ò¡ÆC14
MPOP
AND       M1051F	// L_2nd STEP#15
AND NOT   T4020	// L_2nd SS CLAMP.L UP
AND       T4021	// L_2nd SS CLAMP.L DN
AND NOT   T4022	// L_2nd SS CLAMP.R UP
AND       T4023	// L_2nd SS CLAMP.R DN
AND NOT   T4024	// L_2nd SS SUPPORT DN
AND       T4025	// L_2nd SS SUPPORT UP
AND NOT   T4026	// L_2nd SS SPANKING FW
AND       T4027	// L_2nd SS SPANKING BW
AND NOT   T4028	// L_2nd SS MANDREL FW
AND       T4029	// L_2nd SS MANDREL BW
AND       T4030	// L_2nd SS ALIGN FPCB FW
AND NOT   T4031	// L_2nd SS ALIGN FPCB BW
AND       T4032	// L_2nd SS ALIGN SIDE FW
AND NOT   T4033	// L_2nd SS ALIGN SIDE BW
AND       M04061	// L_2nd_06 Y Pos.2nd SPANK IN
AND       M04070	// L_2nd_07 R Pos.1st IDLE
AND       M04081	// L_2nd_08 T Pos.2nd WORK
AND       P00116	// L_2nd DIE VACUUM EJECTOR ON
OUT       M1053F	// STEP A¢Ò¡ÆC15
// output comment: STEP INITIAL
// output comment: ALIGN FPCB FW [P0122]
// output comment: ALIGN SIDE FW [P0123]
// output comment: L_2nd_08 T Pos.2nd WORK
// output comment: CLAMP.R TOP DN [P0125]
// output comment: SUPPORT DN    [P0124]
// output comment: MANDREL FW      [P0127]
// output comment: L_2nd_07 R Pos.2nd BEND >
// output comment: L_2nd_07 R Pos.3rd BACK >
// output comment: SUPPORT UP     [P0124]           MANDREL BW             [P0127]
// output comment: CLAMP.L TOP DN [P0126]
// output comment: L_2nd_06 Y Pos.2nd SPANK IN >         L_2nd_07 R Pos.1st IDLE >
// output comment: SPANKING FW    [P011C]
// output comment: L_2nd_06 Y Pos.3rd SPANK >
// output comment: L_2nd_06 Y Pos.2nd SPANK IN >
// output comment: SPANKING BW     [P011C]

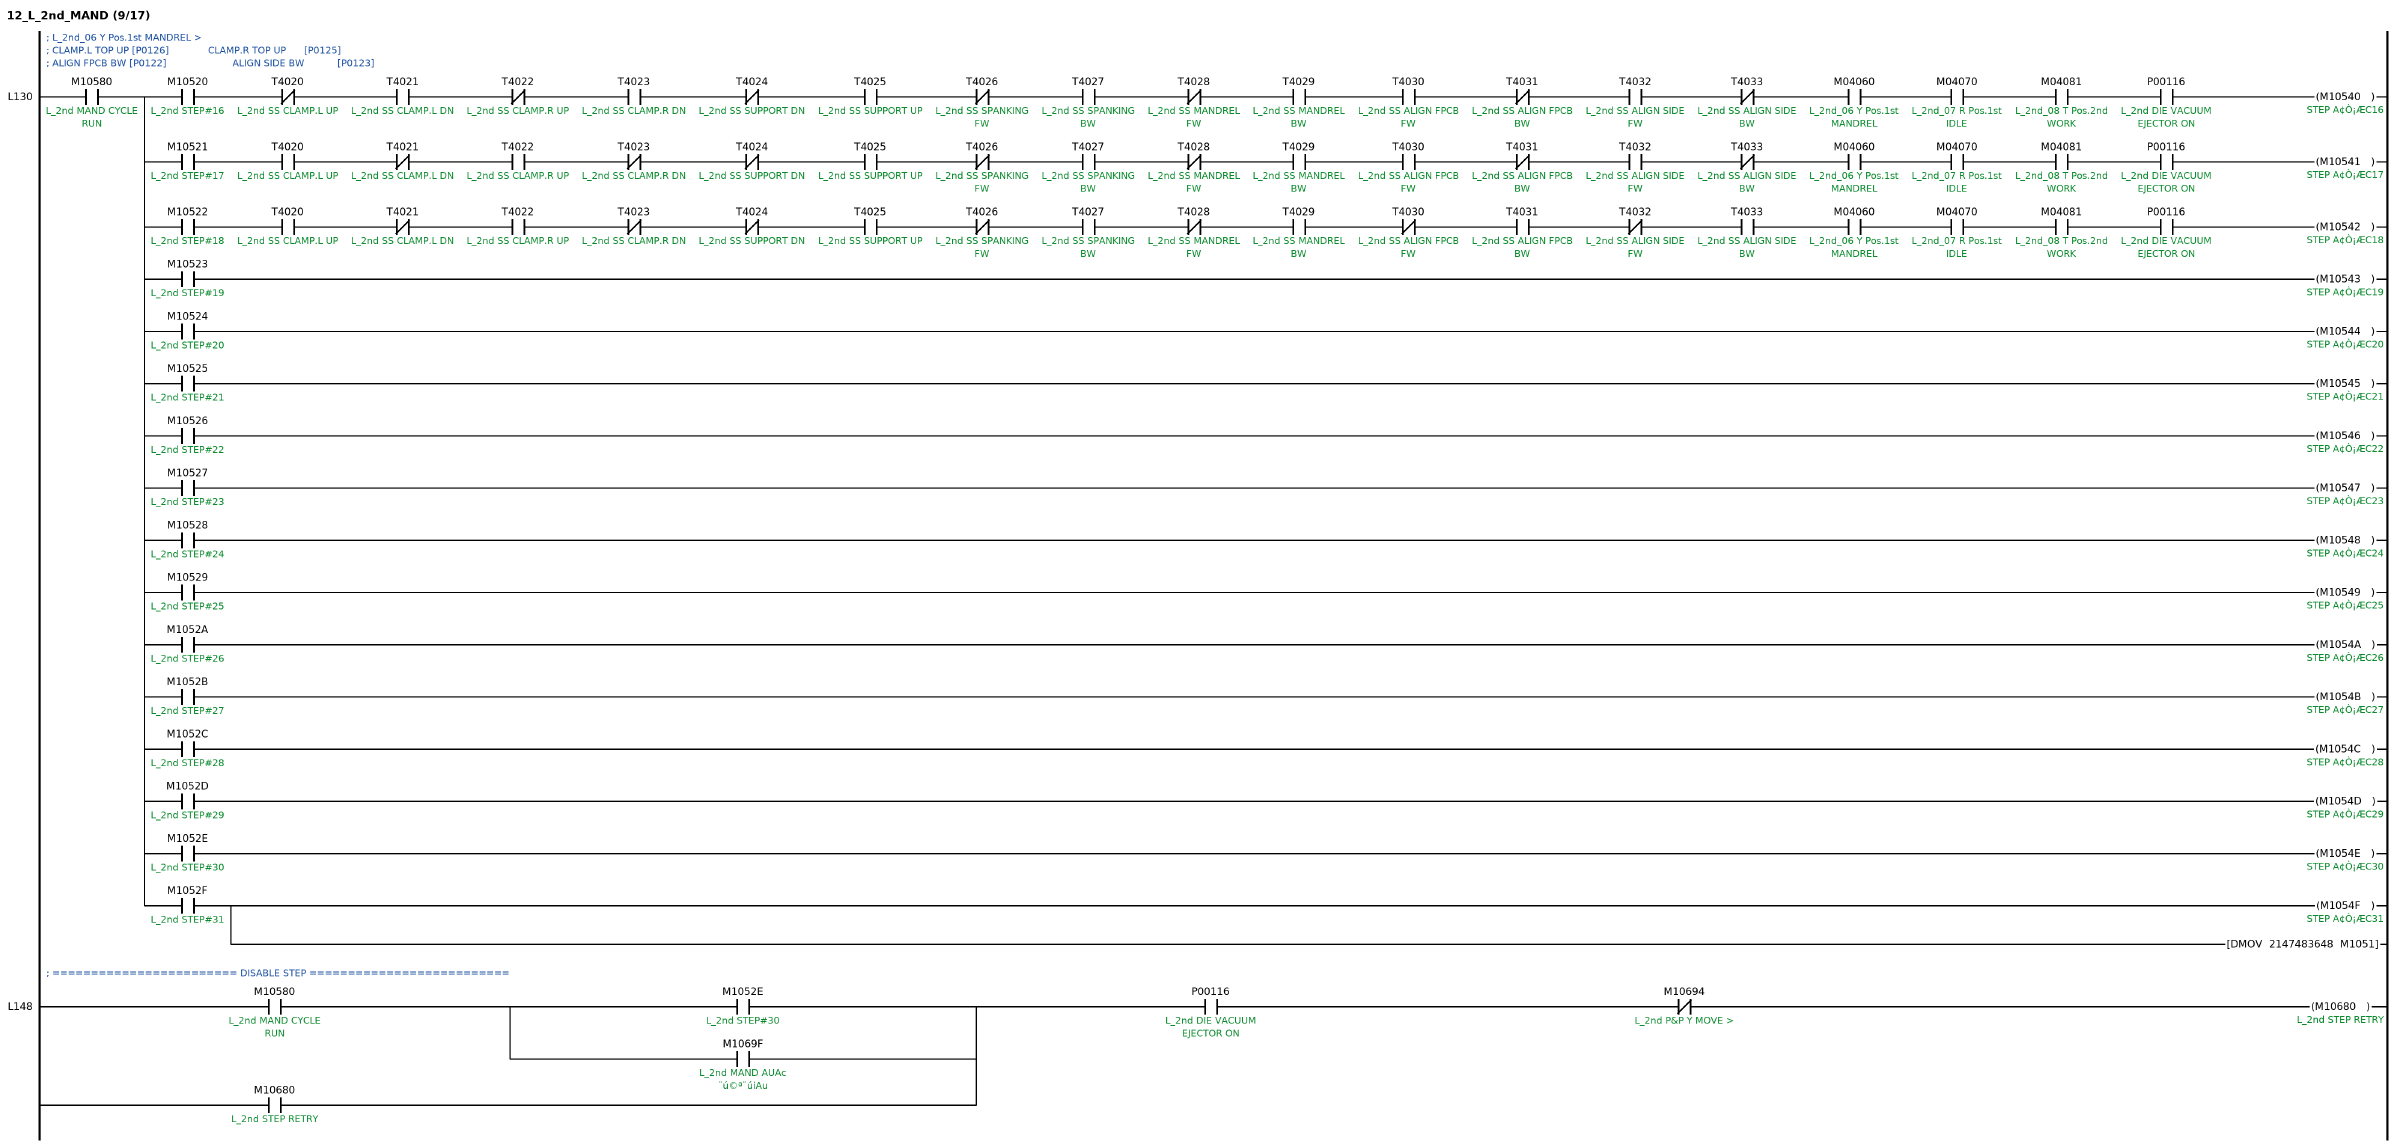
; L130
LOAD      M10580	// L_2nd MAND CYCLE RUN
MPUSH
AND       M10520	// L_2nd STEP#16
AND NOT   T4020	// L_2nd SS CLAMP.L UP
AND       T4021	// L_2nd SS CLAMP.L DN
AND NOT   T4022	// L_2nd SS CLAMP.R UP
AND       T4023	// L_2nd SS CLAMP.R DN
AND NOT   T4024	// L_2nd SS SUPPORT DN
AND       T4025	// L_2nd SS SUPPORT UP
AND NOT   T4026	// L_2nd SS SPANKING FW
AND       T4027	// L_2nd SS SPANKING BW
AND NOT   T4028	// L_2nd SS MANDREL FW
AND       T4029	// L_2nd SS MANDREL BW
AND       T4030	// L_2nd SS ALIGN FPCB FW
AND NOT   T4031	// L_2nd SS ALIGN FPCB BW
AND       T4032	// L_2nd SS ALIGN SIDE FW
AND NOT   T4033	// L_2nd SS ALIGN SIDE BW
AND       M04060	// L_2nd_06 Y Pos.1st MANDREL
AND       M04070	// L_2nd_07 R Pos.1st IDLE
AND       M04081	// L_2nd_08 T Pos.2nd WORK
AND       P00116	// L_2nd DIE VACUUM EJECTOR ON
OUT       M10540	// STEP A¢Ò¡ÆC16
MLOAD
AND       M10521	// L_2nd STEP#17
AND       T4020	// L_2nd SS CLAMP.L UP
AND NOT   T4021	// L_2nd SS CLAMP.L DN
AND       T4022	// L_2nd SS CLAMP.R UP
AND NOT   T4023	// L_2nd SS CLAMP.R DN
AND NOT   T4024	// L_2nd SS SUPPORT DN
AND       T4025	// L_2nd SS SUPPORT UP
AND NOT   T4026	// L_2nd SS SPANKING FW
AND       T4027	// L_2nd SS SPANKING BW
AND NOT   T4028	// L_2nd SS MANDREL FW
AND       T4029	// L_2nd SS MANDREL BW
AND       T4030	// L_2nd SS ALIGN FPCB FW
AND NOT   T4031	// L_2nd SS ALIGN FPCB BW
AND       T4032	// L_2nd SS ALIGN SIDE FW
AND NOT   T4033	// L_2nd SS ALIGN SIDE BW
AND       M04060	// L_2nd_06 Y Pos.1st MANDREL
AND       M04070	// L_2nd_07 R Pos.1st IDLE
AND       M04081	// L_2nd_08 T Pos.2nd WORK
AND       P00116	// L_2nd DIE VACUUM EJECTOR ON
OUT       M10541	// STEP A¢Ò¡ÆC17
MLOAD
AND       M10522	// L_2nd STEP#18
AND       T4020	// L_2nd SS CLAMP.L UP
AND NOT   T4021	// L_2nd SS CLAMP.L DN
AND       T4022	// L_2nd SS CLAMP.R UP
AND NOT   T4023	// L_2nd SS CLAMP.R DN
AND NOT   T4024	// L_2nd SS SUPPORT DN
AND       T4025	// L_2nd SS SUPPORT UP
AND NOT   T4026	// L_2nd SS SPANKING FW
AND       T4027	// L_2nd SS SPANKING BW
AND NOT   T4028	// L_2nd SS MANDREL FW
AND       T4029	// L_2nd SS MANDREL BW
AND NOT   T4030	// L_2nd SS ALIGN FPCB FW
AND       T4031	// L_2nd SS ALIGN FPCB BW
AND NOT   T4032	// L_2nd SS ALIGN SIDE FW
AND       T4033	// L_2nd SS ALIGN SIDE BW
AND       M04060	// L_2nd_06 Y Pos.1st MANDREL
AND       M04070	// L_2nd_07 R Pos.1st IDLE
AND       M04081	// L_2nd_08 T Pos.2nd WORK
AND       P00116	// L_2nd DIE VACUUM EJECTOR ON
OUT       M10542	// STEP A¢Ò¡ÆC18
MLOAD
AND       M10523	// L_2nd STEP#19
OUT       M10543	// STEP A¢Ò¡ÆC19
MLOAD
AND       M10524	// L_2nd STEP#20
OUT       M10544	// STEP A¢Ò¡ÆC20
MLOAD
AND       M10525	// L_2nd STEP#21
OUT       M10545	// STEP A¢Ò¡ÆC21
MLOAD
AND       M10526	// L_2nd STEP#22
OUT       M10546	// STEP A¢Ò¡ÆC22
MLOAD
AND       M10527	// L_2nd STEP#23
OUT       M10547	// STEP A¢Ò¡ÆC23
MLOAD
AND       M10528	// L_2nd STEP#24
OUT       M10548	// STEP A¢Ò¡ÆC24
MLOAD
AND       M10529	// L_2nd STEP#25
OUT       M10549	// STEP A¢Ò¡ÆC25
MLOAD
AND       M1052A	// L_2nd STEP#26
OUT       M1054A	// STEP A¢Ò¡ÆC26
MLOAD
AND       M1052B	// L_2nd STEP#27
OUT       M1054B	// STEP A¢Ò¡ÆC27
MLOAD
AND       M1052C	// L_2nd STEP#28
OUT       M1054C	// STEP A¢Ò¡ÆC28
MLOAD
AND       M1052D	// L_2nd STEP#29
OUT       M1054D	// STEP A¢Ò¡ÆC29
MLOAD
AND       M1052E	// L_2nd STEP#30
OUT       M1054E	// STEP A¢Ò¡ÆC30
MPOP
AND       M1052F	// L_2nd STEP#31
OUT       M1054F	// STEP A¢Ò¡ÆC31
DMOV      2147483648 M1051
// output comment: L_2nd_06 Y Pos.1st MANDREL >
// output comment: CLAMP.L TOP UP [P0126]             CLAMP.R TOP UP      [P0125]
// output comment: ALIGN FPCB BW [P0122]                      ALIGN SIDE BW           [P0123]
// ======================== DISABLE STEP ==========================
; L148
LOAD      M10580	// L_2nd MAND CYCLE RUN
LOAD      M1052E	// L_2nd STEP#30
OR        M1069F	// L_2nd MAND AUAc ¨ú©ª¨úiAu
AND LOAD
OR        M10680	// L_2nd STEP RETRY
AND       P00116	// L_2nd DIE VACUUM EJECTOR ON
AND NOT   M10694	// L_2nd P&P Y MOVE >
OUT       M10680	// L_2nd STEP RETRY

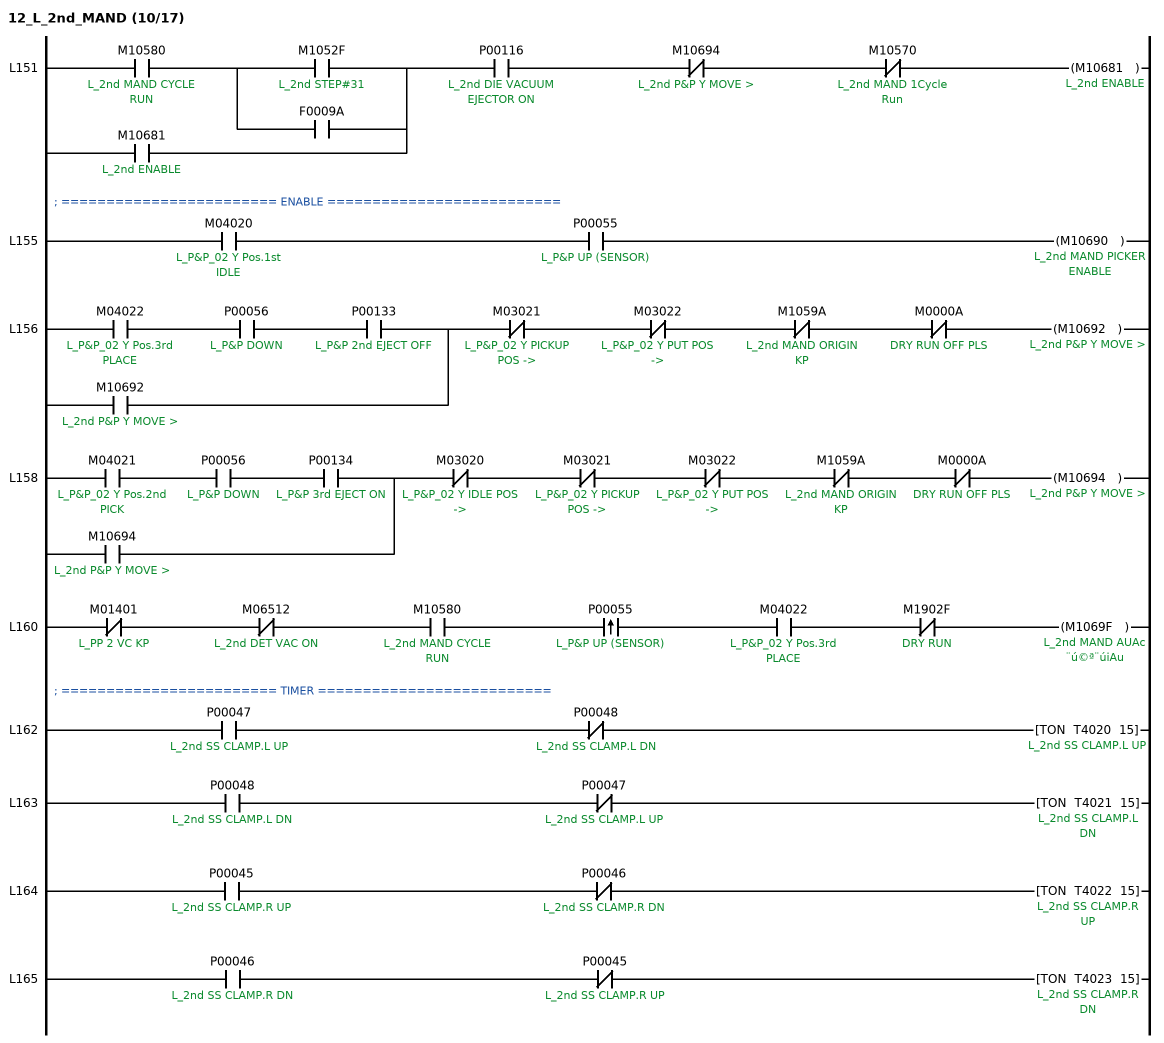
; L151
LOAD      M10580	// L_2nd MAND CYCLE RUN
LOAD      M1052F	// L_2nd STEP#31
OR        F0009A
AND LOAD
OR        M10681	// L_2nd ENABLE
AND       P00116	// L_2nd DIE VACUUM EJECTOR ON
AND NOT   M10694	// L_2nd P&P Y MOVE >
AND NOT   M10570	// L_2nd MAND 1Cycle Run
OUT       M10681	// L_2nd ENABLE
// ======================== ENABLE ==========================
; L155
LOAD      M04020	// L_P&P_02 Y Pos.1st IDLE
AND       P00055	// L_P&P UP (SENSOR)
OUT       M10690	// L_2nd MAND PICKER ENABLE
; L156
LOAD      M04022	// L_P&P_02 Y Pos.3rd PLACE
AND       P00056	// L_P&P DOWN
AND       P00133	// L_P&P 2nd EJECT OFF
OR        M10692	// L_2nd P&P Y MOVE >
AND NOT   M03021	// L_P&P_02 Y PICKUP POS ->
AND NOT   M03022	// L_P&P_02 Y PUT POS ->
AND NOT   M1059A	// L_2nd MAND ORIGIN KP
AND NOT   M0000A	// DRY RUN OFF PLS
OUT       M10692	// L_2nd P&P Y MOVE >
; L158
LOAD      M04021	// L_P&P_02 Y Pos.2nd PICK
AND       P00056	// L_P&P DOWN
AND       P00134	// L_P&P 3rd EJECT ON
OR        M10694	// L_2nd P&P Y MOVE >
AND NOT   M03020	// L_P&P_02 Y IDLE POS ->
AND NOT   M03021	// L_P&P_02 Y PICKUP POS ->
AND NOT   M03022	// L_P&P_02 Y PUT POS ->
AND NOT   M1059A	// L_2nd MAND ORIGIN KP
AND NOT   M0000A	// DRY RUN OFF PLS
OUT       M10694	// L_2nd P&P Y MOVE >
; L160
LOAD NOT  M01401	// L_PP 2 VC KP
AND NOT   M06512	// L_2nd DET VAC ON
AND       M10580	// L_2nd MAND CYCLE RUN
ANDP      P00055	// L_P&P UP (SENSOR)
AND       M04022	// L_P&P_02 Y Pos.3rd PLACE
AND NOT   M1902F	// DRY RUN
OUT       M1069F	// L_2nd MAND AUAc ¨ú©ª¨úiAu
// ======================== TIMER ==========================
; L162
LOAD      P00047	// L_2nd SS CLAMP.L UP
AND NOT   P00048	// L_2nd SS CLAMP.L DN
TON       T4020 15	// L_2nd SS CLAMP.L UP
; L163
LOAD      P00048	// L_2nd SS CLAMP.L DN
AND NOT   P00047	// L_2nd SS CLAMP.L UP
TON       T4021 15	// L_2nd SS CLAMP.L DN
; L164
LOAD      P00045	// L_2nd SS CLAMP.R UP
AND NOT   P00046	// L_2nd SS CLAMP.R DN
TON       T4022 15	// L_2nd SS CLAMP.R UP
; L165
LOAD      P00046	// L_2nd SS CLAMP.R DN
AND NOT   P00045	// L_2nd SS CLAMP.R UP
TON       T4023 15	// L_2nd SS CLAMP.R DN

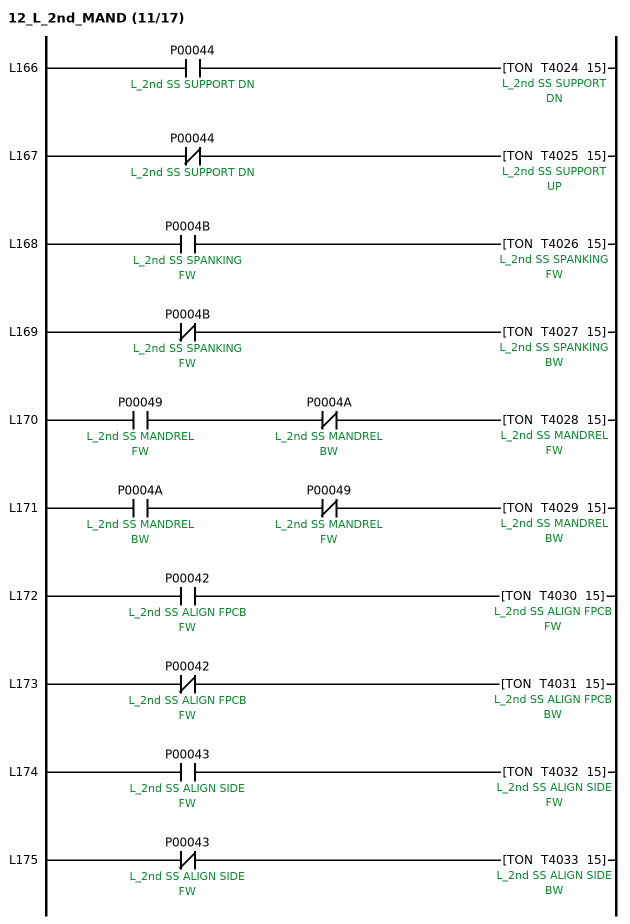
; L166
LOAD      P00044	// L_2nd SS SUPPORT DN
TON       T4024 15	// L_2nd SS SUPPORT DN
; L167
LOAD NOT  P00044	// L_2nd SS SUPPORT DN
TON       T4025 15	// L_2nd SS SUPPORT UP
; L168
LOAD      P0004B	// L_2nd SS SPANKING FW
TON       T4026 15	// L_2nd SS SPANKING FW
; L169
LOAD NOT  P0004B	// L_2nd SS SPANKING FW
TON       T4027 15	// L_2nd SS SPANKING BW
; L170
LOAD      P00049	// L_2nd SS MANDREL FW
AND NOT   P0004A	// L_2nd SS MANDREL BW
TON       T4028 15	// L_2nd SS MANDREL FW
; L171
LOAD      P0004A	// L_2nd SS MANDREL BW
AND NOT   P00049	// L_2nd SS MANDREL FW
TON       T4029 15	// L_2nd SS MANDREL BW
; L172
LOAD      P00042	// L_2nd SS ALIGN FPCB FW
TON       T4030 15	// L_2nd SS ALIGN FPCB FW
; L173
LOAD NOT  P00042	// L_2nd SS ALIGN FPCB FW
TON       T4031 15	// L_2nd SS ALIGN FPCB BW
; L174
LOAD      P00043	// L_2nd SS ALIGN SIDE FW
TON       T4032 15	// L_2nd SS ALIGN SIDE FW
; L175
LOAD NOT  P00043	// L_2nd SS ALIGN SIDE FW
TON       T4033 15	// L_2nd SS ALIGN SIDE BW

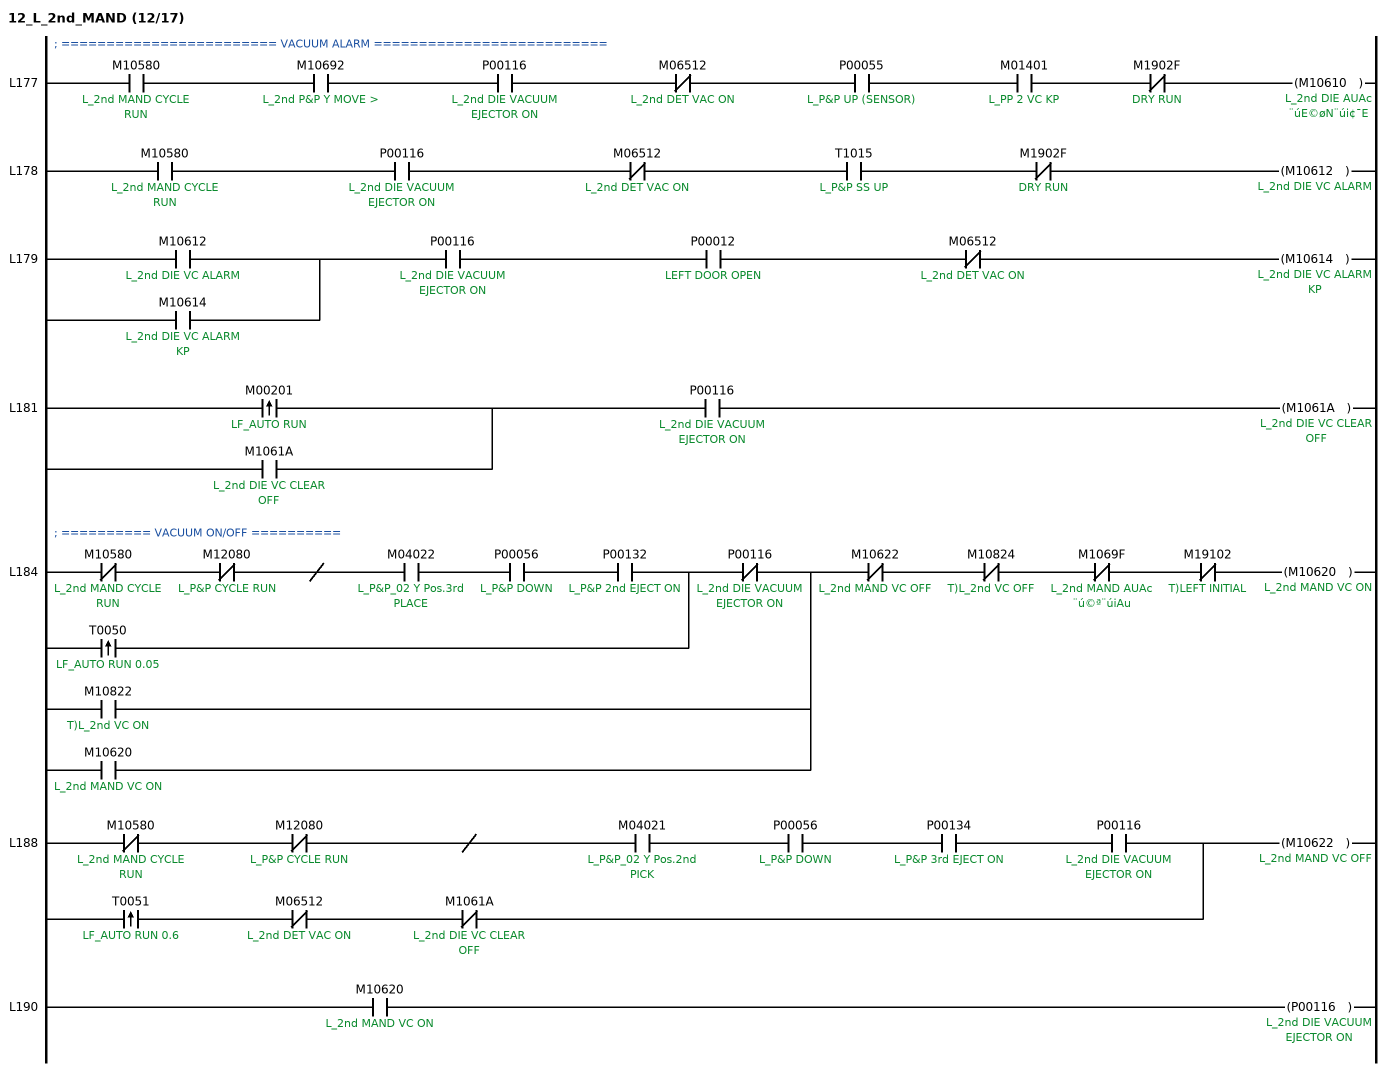
// ======================== VACUUM ALARM ==========================
; L177
LOAD      M10580	// L_2nd MAND CYCLE RUN
AND       M10692	// L_2nd P&P Y MOVE >
AND       P00116	// L_2nd DIE VACUUM EJECTOR ON
AND NOT   M06512	// L_2nd DET VAC ON
AND       P00055	// L_P&P UP (SENSOR)
AND       M01401	// L_PP 2 VC KP
AND NOT   M1902F	// DRY RUN
OUT       M10610	// L_2nd DIE AUAc ¨úE©øN¨úi¢¯E
; L178
LOAD      M10580	// L_2nd MAND CYCLE RUN
AND       P00116	// L_2nd DIE VACUUM EJECTOR ON
AND NOT   M06512	// L_2nd DET VAC ON
AND       T1015	// L_P&P SS UP
AND NOT   M1902F	// DRY RUN
OUT       M10612	// L_2nd DIE VC ALARM
; L179
LOAD      M10612	// L_2nd DIE VC ALARM
OR        M10614	// L_2nd DIE VC ALARM KP
AND       P00116	// L_2nd DIE VACUUM EJECTOR ON
AND       P00012	// LEFT DOOR OPEN
AND NOT   M06512	// L_2nd DET VAC ON
OUT       M10614	// L_2nd DIE VC ALARM KP
; L181
LOADP     M00201	// LF_AUTO RUN
OR        M1061A	// L_2nd DIE VC CLEAR OFF
AND       P00116	// L_2nd DIE VACUUM EJECTOR ON
OUT       M1061A	// L_2nd DIE VC CLEAR OFF
// ========== VACUUM ON/OFF ==========
; L184
LOAD NOT  M10580	// L_2nd MAND CYCLE RUN
AND NOT   M12080	// L_P&P CYCLE RUN
NOT
AND       M04022	// L_P&P_02 Y Pos.3rd PLACE
AND       P00056	// L_P&P DOWN
AND       P00132	// L_P&P 2nd EJECT ON
ORP       T0050	// LF_AUTO RUN 0.05
AND NOT   P00116	// L_2nd DIE VACUUM EJECTOR ON
OR        M10822	// T)L_2nd VC ON
OR        M10620	// L_2nd MAND VC ON
AND NOT   M10622	// L_2nd MAND VC OFF
AND NOT   M10824	// T)L_2nd VC OFF
AND NOT   M1069F	// L_2nd MAND AUAc ¨ú©ª¨úiAu
AND NOT   M19102	// T)LEFT INITIAL
OUT       M10620	// L_2nd MAND VC ON
; L188
LOAD NOT  M10580	// L_2nd MAND CYCLE RUN
AND NOT   M12080	// L_P&P CYCLE RUN
NOT
AND       M04021	// L_P&P_02 Y Pos.2nd PICK
AND       P00056	// L_P&P DOWN
AND       P00134	// L_P&P 3rd EJECT ON
AND       P00116	// L_2nd DIE VACUUM EJECTOR ON
LOADP     T0051	// LF_AUTO RUN 0.6
AND NOT   M06512	// L_2nd DET VAC ON
AND NOT   M1061A	// L_2nd DIE VC CLEAR OFF
OR LOAD
OUT       M10622	// L_2nd MAND VC OFF
; L190
LOAD      M10620	// L_2nd MAND VC ON
OUT       P00116	// L_2nd DIE VACUUM EJECTOR ON

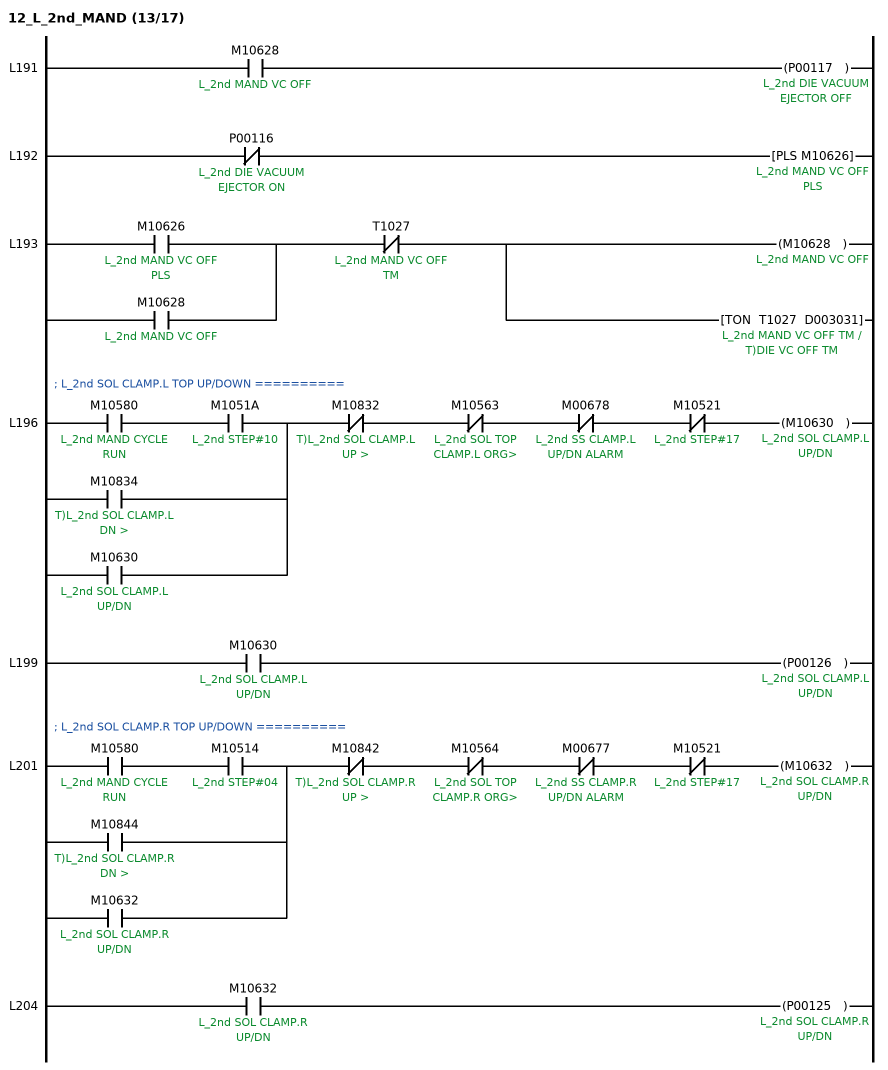
; L191
LOAD      M10628	// L_2nd MAND VC OFF
OUT       P00117	// L_2nd DIE VACUUM EJECTOR OFF
; L192
LOAD NOT  P00116	// L_2nd DIE VACUUM EJECTOR ON
OUTP      M10626	// L_2nd MAND VC OFF PLS
; L193
LOAD      M10626	// L_2nd MAND VC OFF PLS
OR        M10628	// L_2nd MAND VC OFF
AND NOT   T1027	// L_2nd MAND VC OFF TM
OUT       M10628	// L_2nd MAND VC OFF
TON       T1027 D003031	// L_2nd MAND VC OFF TM / T)DIE VC OFF TM
// L_2nd SOL CLAMP.L TOP UP/DOWN ==========
; L196
LOAD      M10580	// L_2nd MAND CYCLE RUN
AND       M1051A	// L_2nd STEP#10
OR        M10834	// T)L_2nd SOL CLAMP.L DN >
OR        M10630	// L_2nd SOL CLAMP.L UP/DN
AND NOT   M10832	// T)L_2nd SOL CLAMP.L UP >
AND NOT   M10563	// L_2nd SOL TOP CLAMP.L ORG>
AND NOT   M00678	// L_2nd SS CLAMP.L UP/DN ALARM
AND NOT   M10521	// L_2nd STEP#17
OUT       M10630	// L_2nd SOL CLAMP.L UP/DN
; L199
LOAD      M10630	// L_2nd SOL CLAMP.L UP/DN
OUT       P00126	// L_2nd SOL CLAMP.L UP/DN
// L_2nd SOL CLAMP.R TOP UP/DOWN ==========
; L201
LOAD      M10580	// L_2nd MAND CYCLE RUN
AND       M10514	// L_2nd STEP#04
OR        M10844	// T)L_2nd SOL CLAMP.R DN >
OR        M10632	// L_2nd SOL CLAMP.R UP/DN
AND NOT   M10842	// T)L_2nd SOL CLAMP.R UP >
AND NOT   M10564	// L_2nd SOL TOP CLAMP.R ORG>
AND NOT   M00677	// L_2nd SS CLAMP.R UP/DN ALARM
AND NOT   M10521	// L_2nd STEP#17
OUT       M10632	// L_2nd SOL CLAMP.R UP/DN
; L204
LOAD      M10632	// L_2nd SOL CLAMP.R UP/DN
OUT       P00125	// L_2nd SOL CLAMP.R UP/DN

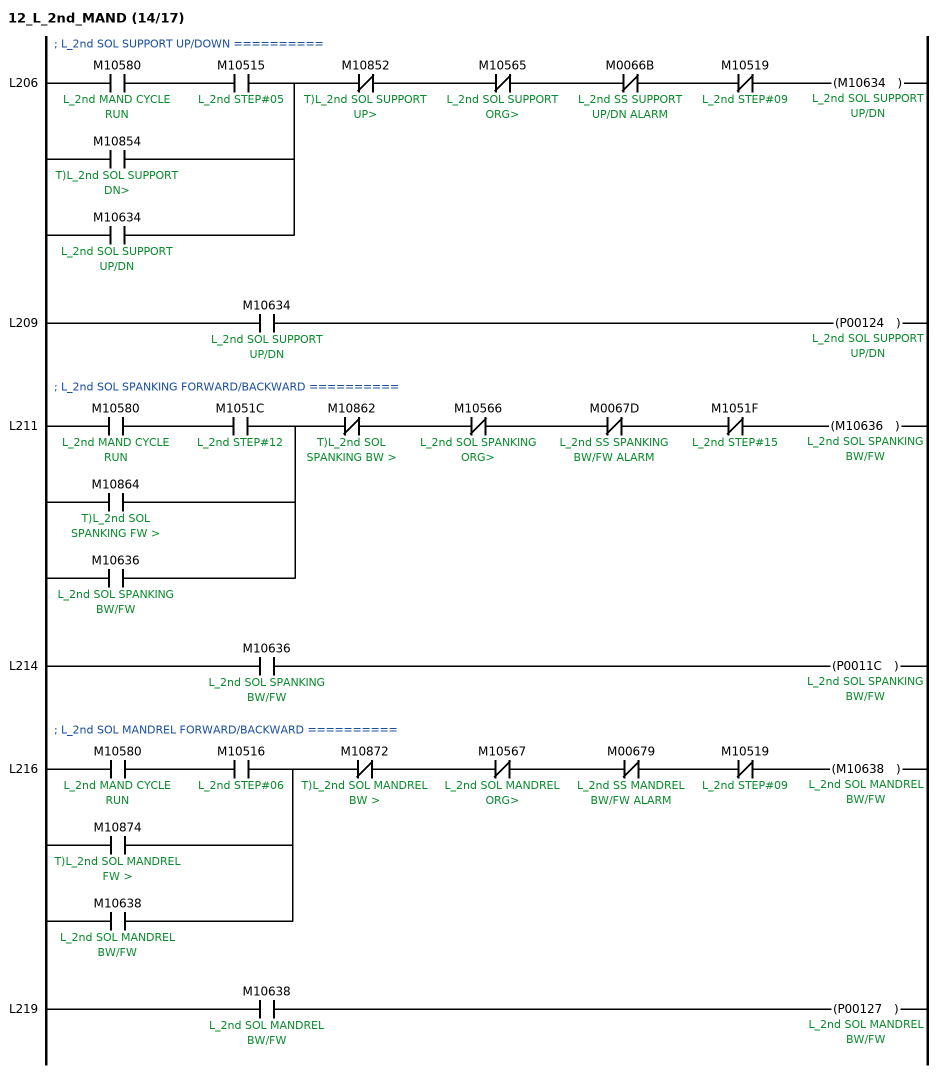
// L_2nd SOL SUPPORT UP/DOWN ==========
; L206
LOAD      M10580	// L_2nd MAND CYCLE RUN
AND       M10515	// L_2nd STEP#05
OR        M10854	// T)L_2nd SOL SUPPORT DN>
OR        M10634	// L_2nd SOL SUPPORT UP/DN
AND NOT   M10852	// T)L_2nd SOL SUPPORT UP>
AND NOT   M10565	// L_2nd SOL SUPPORT ORG>
AND NOT   M0066B	// L_2nd SS SUPPORT UP/DN ALARM
AND NOT   M10519	// L_2nd STEP#09
OUT       M10634	// L_2nd SOL SUPPORT UP/DN
; L209
LOAD      M10634	// L_2nd SOL SUPPORT UP/DN
OUT       P00124	// L_2nd SOL SUPPORT UP/DN
// L_2nd SOL SPANKING FORWARD/BACKWARD ==========
; L211
LOAD      M10580	// L_2nd MAND CYCLE RUN
AND       M1051C	// L_2nd STEP#12
OR        M10864	// T)L_2nd SOL SPANKING FW >
OR        M10636	// L_2nd SOL SPANKING BW/FW
AND NOT   M10862	// T)L_2nd SOL SPANKING BW >
AND NOT   M10566	// L_2nd SOL SPANKING ORG>
AND NOT   M0067D	// L_2nd SS SPANKING BW/FW ALARM
AND NOT   M1051F	// L_2nd STEP#15
OUT       M10636	// L_2nd SOL SPANKING BW/FW
; L214
LOAD      M10636	// L_2nd SOL SPANKING BW/FW
OUT       P0011C	// L_2nd SOL SPANKING BW/FW
// L_2nd SOL MANDREL FORWARD/BACKWARD ==========
; L216
LOAD      M10580	// L_2nd MAND CYCLE RUN
AND       M10516	// L_2nd STEP#06
OR        M10874	// T)L_2nd SOL MANDREL FW >
OR        M10638	// L_2nd SOL MANDREL BW/FW
AND NOT   M10872	// T)L_2nd SOL MANDREL BW >
AND NOT   M10567	// L_2nd SOL MANDREL ORG>
AND NOT   M00679	// L_2nd SS MANDREL BW/FW ALARM
AND NOT   M10519	// L_2nd STEP#09
OUT       M10638	// L_2nd SOL MANDREL BW/FW
; L219
LOAD      M10638	// L_2nd SOL MANDREL BW/FW
OUT       P00127	// L_2nd SOL MANDREL BW/FW

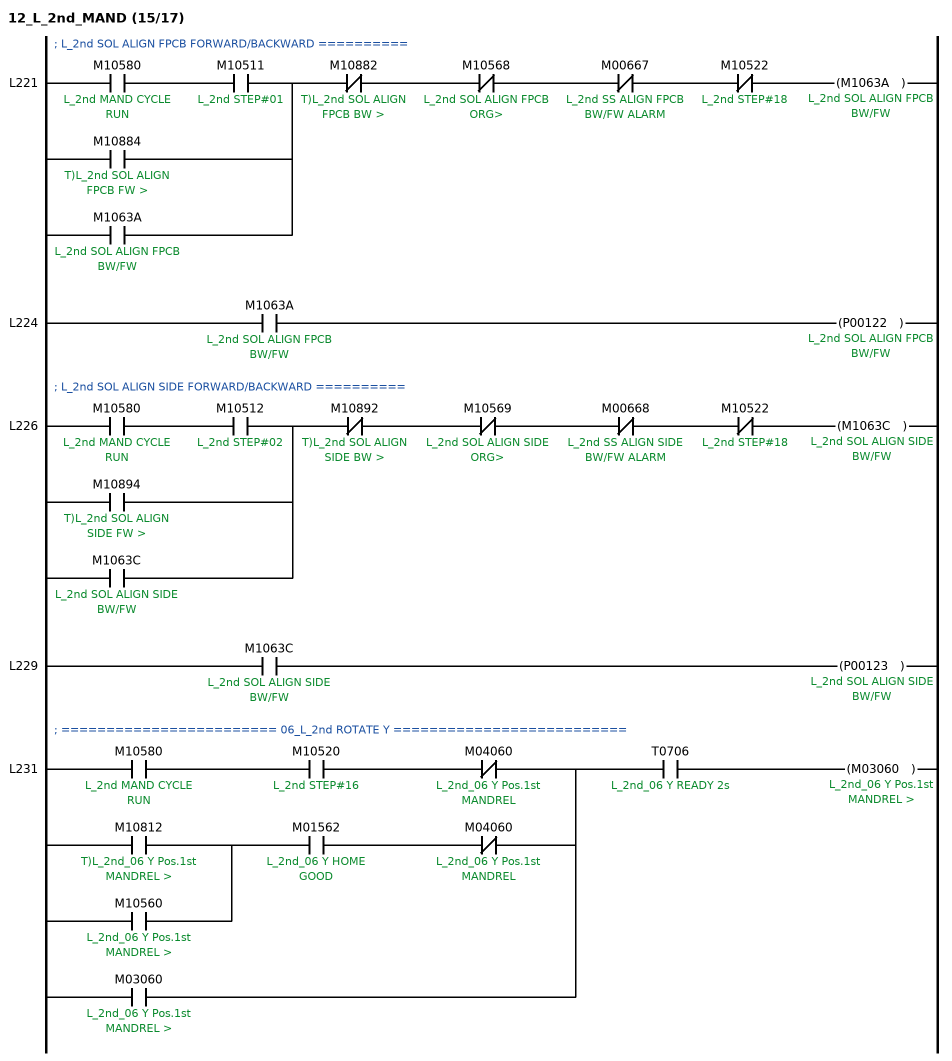
// L_2nd SOL ALIGN FPCB FORWARD/BACKWARD ==========
; L221
LOAD      M10580	// L_2nd MAND CYCLE RUN
AND       M10511	// L_2nd STEP#01
OR        M10884	// T)L_2nd SOL ALIGN FPCB FW >
OR        M1063A	// L_2nd SOL ALIGN FPCB BW/FW
AND NOT   M10882	// T)L_2nd SOL ALIGN FPCB BW >
AND NOT   M10568	// L_2nd SOL ALIGN FPCB ORG>
AND NOT   M00667	// L_2nd SS ALIGN FPCB BW/FW ALARM
AND NOT   M10522	// L_2nd STEP#18
OUT       M1063A	// L_2nd SOL ALIGN FPCB BW/FW
; L224
LOAD      M1063A	// L_2nd SOL ALIGN FPCB BW/FW
OUT       P00122	// L_2nd SOL ALIGN FPCB BW/FW
// L_2nd SOL ALIGN SIDE FORWARD/BACKWARD ==========
; L226
LOAD      M10580	// L_2nd MAND CYCLE RUN
AND       M10512	// L_2nd STEP#02
OR        M10894	// T)L_2nd SOL ALIGN SIDE FW >
OR        M1063C	// L_2nd SOL ALIGN SIDE BW/FW
AND NOT   M10892	// T)L_2nd SOL ALIGN SIDE BW >
AND NOT   M10569	// L_2nd SOL ALIGN SIDE ORG>
AND NOT   M00668	// L_2nd SS ALIGN SIDE BW/FW ALARM
AND NOT   M10522	// L_2nd STEP#18
OUT       M1063C	// L_2nd SOL ALIGN SIDE BW/FW
; L229
LOAD      M1063C	// L_2nd SOL ALIGN SIDE BW/FW
OUT       P00123	// L_2nd SOL ALIGN SIDE BW/FW
// ======================== 06_L_2nd ROTATE Y ==========================
; L231
LOAD      M10580	// L_2nd MAND CYCLE RUN
AND       M10520	// L_2nd STEP#16
AND NOT   M04060	// L_2nd_06 Y Pos.1st MANDREL
LOAD      M10812	// T)L_2nd_06 Y Pos.1st MANDREL >
OR        M10560	// L_2nd_06 Y Pos.1st MANDREL >
AND       M01562	// L_2nd_06 Y HOME GOOD
AND NOT   M04060	// L_2nd_06 Y Pos.1st MANDREL
OR LOAD
OR        M03060	// L_2nd_06 Y Pos.1st MANDREL >
AND       T0706	// L_2nd_06 Y READY 2s
OUT       M03060	// L_2nd_06 Y Pos.1st MANDREL >

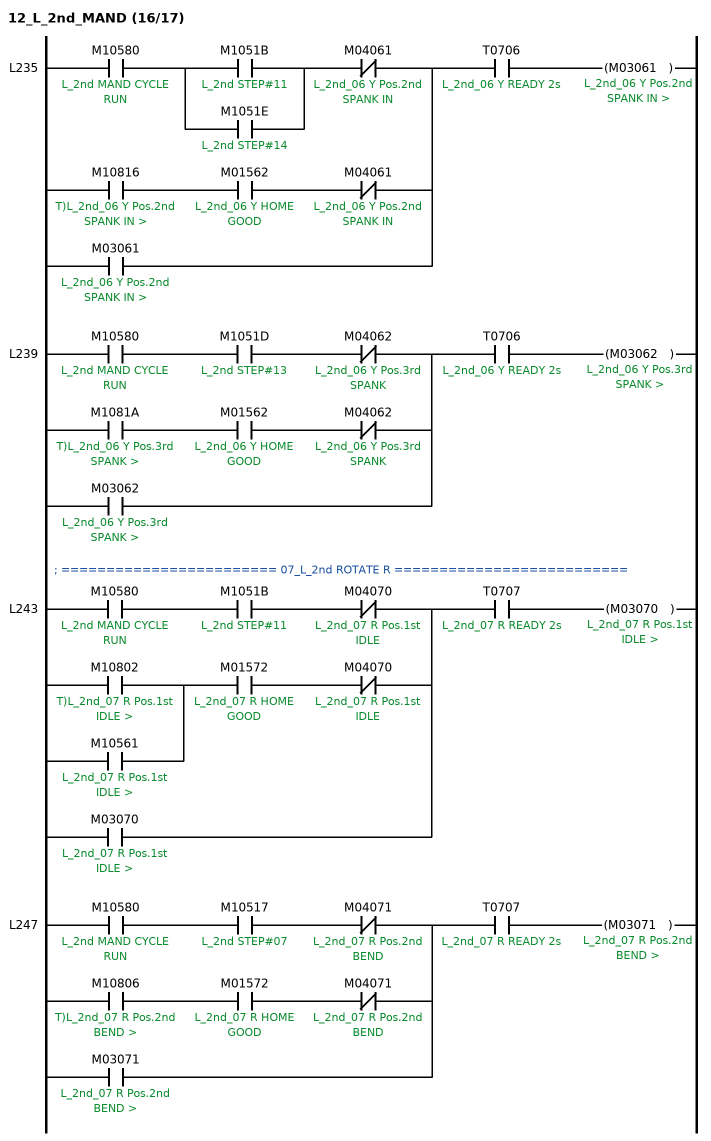
; L235
LOAD      M10580	// L_2nd MAND CYCLE RUN
LOAD      M1051B	// L_2nd STEP#11
OR        M1051E	// L_2nd STEP#14
AND LOAD
AND NOT   M04061	// L_2nd_06 Y Pos.2nd SPANK IN
LOAD      M10816	// T)L_2nd_06 Y Pos.2nd SPANK IN >
AND       M01562	// L_2nd_06 Y HOME GOOD
AND NOT   M04061	// L_2nd_06 Y Pos.2nd SPANK IN
OR LOAD
OR        M03061	// L_2nd_06 Y Pos.2nd SPANK IN >
AND       T0706	// L_2nd_06 Y READY 2s
OUT       M03061	// L_2nd_06 Y Pos.2nd SPANK IN >
; L239
LOAD      M10580	// L_2nd MAND CYCLE RUN
AND       M1051D	// L_2nd STEP#13
AND NOT   M04062	// L_2nd_06 Y Pos.3rd SPANK
LOAD      M1081A	// T)L_2nd_06 Y Pos.3rd SPANK >
AND       M01562	// L_2nd_06 Y HOME GOOD
AND NOT   M04062	// L_2nd_06 Y Pos.3rd SPANK
OR LOAD
OR        M03062	// L_2nd_06 Y Pos.3rd SPANK >
AND       T0706	// L_2nd_06 Y READY 2s
OUT       M03062	// L_2nd_06 Y Pos.3rd SPANK >
// ======================== 07_L_2nd ROTATE R ==========================
; L243
LOAD      M10580	// L_2nd MAND CYCLE RUN
AND       M1051B	// L_2nd STEP#11
AND NOT   M04070	// L_2nd_07 R Pos.1st IDLE
LOAD      M10802	// T)L_2nd_07 R Pos.1st IDLE >
OR        M10561	// L_2nd_07 R Pos.1st IDLE >
AND       M01572	// L_2nd_07 R HOME GOOD
AND NOT   M04070	// L_2nd_07 R Pos.1st IDLE
OR LOAD
OR        M03070	// L_2nd_07 R Pos.1st IDLE >
AND       T0707	// L_2nd_07 R READY 2s
OUT       M03070	// L_2nd_07 R Pos.1st IDLE >
; L247
LOAD      M10580	// L_2nd MAND CYCLE RUN
AND       M10517	// L_2nd STEP#07
AND NOT   M04071	// L_2nd_07 R Pos.2nd BEND
LOAD      M10806	// T)L_2nd_07 R Pos.2nd BEND >
AND       M01572	// L_2nd_07 R HOME GOOD
AND NOT   M04071	// L_2nd_07 R Pos.2nd BEND
OR LOAD
OR        M03071	// L_2nd_07 R Pos.2nd BEND >
AND       T0707	// L_2nd_07 R READY 2s
OUT       M03071	// L_2nd_07 R Pos.2nd BEND >

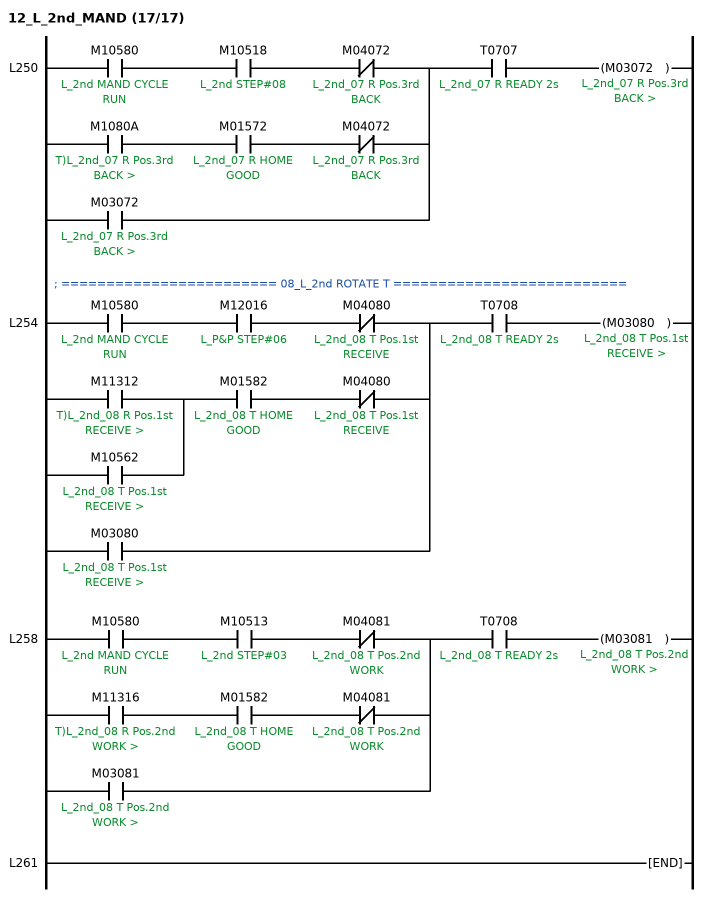
; L250
LOAD      M10580	// L_2nd MAND CYCLE RUN
AND       M10518	// L_2nd STEP#08
AND NOT   M04072	// L_2nd_07 R Pos.3rd BACK
LOAD      M1080A	// T)L_2nd_07 R Pos.3rd BACK >
AND       M01572	// L_2nd_07 R HOME GOOD
AND NOT   M04072	// L_2nd_07 R Pos.3rd BACK
OR LOAD
OR        M03072	// L_2nd_07 R Pos.3rd BACK >
AND       T0707	// L_2nd_07 R READY 2s
OUT       M03072	// L_2nd_07 R Pos.3rd BACK >
// ======================== 08_L_2nd ROTATE T ==========================
; L254
LOAD      M10580	// L_2nd MAND CYCLE RUN
AND       M12016	// L_P&P STEP#06
AND NOT   M04080	// L_2nd_08 T Pos.1st RECEIVE
LOAD      M11312	// T)L_2nd_08 R Pos.1st RECEIVE >
OR        M10562	// L_2nd_08 T Pos.1st RECEIVE >
AND       M01582	// L_2nd_08 T HOME GOOD
AND NOT   M04080	// L_2nd_08 T Pos.1st RECEIVE
OR LOAD
OR        M03080	// L_2nd_08 T Pos.1st RECEIVE >
AND       T0708	// L_2nd_08 T READY 2s
OUT       M03080	// L_2nd_08 T Pos.1st RECEIVE >
; L258
LOAD      M10580	// L_2nd MAND CYCLE RUN
AND       M10513	// L_2nd STEP#03
AND NOT   M04081	// L_2nd_08 T Pos.2nd WORK
LOAD      M11316	// T)L_2nd_08 R Pos.2nd WORK >
AND       M01582	// L_2nd_08 T HOME GOOD
AND NOT   M04081	// L_2nd_08 T Pos.2nd WORK
OR LOAD
OR        M03081	// L_2nd_08 T Pos.2nd WORK >
AND       T0708	// L_2nd_08 T READY 2s
OUT       M03081	// L_2nd_08 T Pos.2nd WORK >
; L261
END

PROGRAM 13_L_3rd_MAND (task: ¨ö¨¬A¥ì CA¡¤I¡¾¡¿¡¤¡Í)

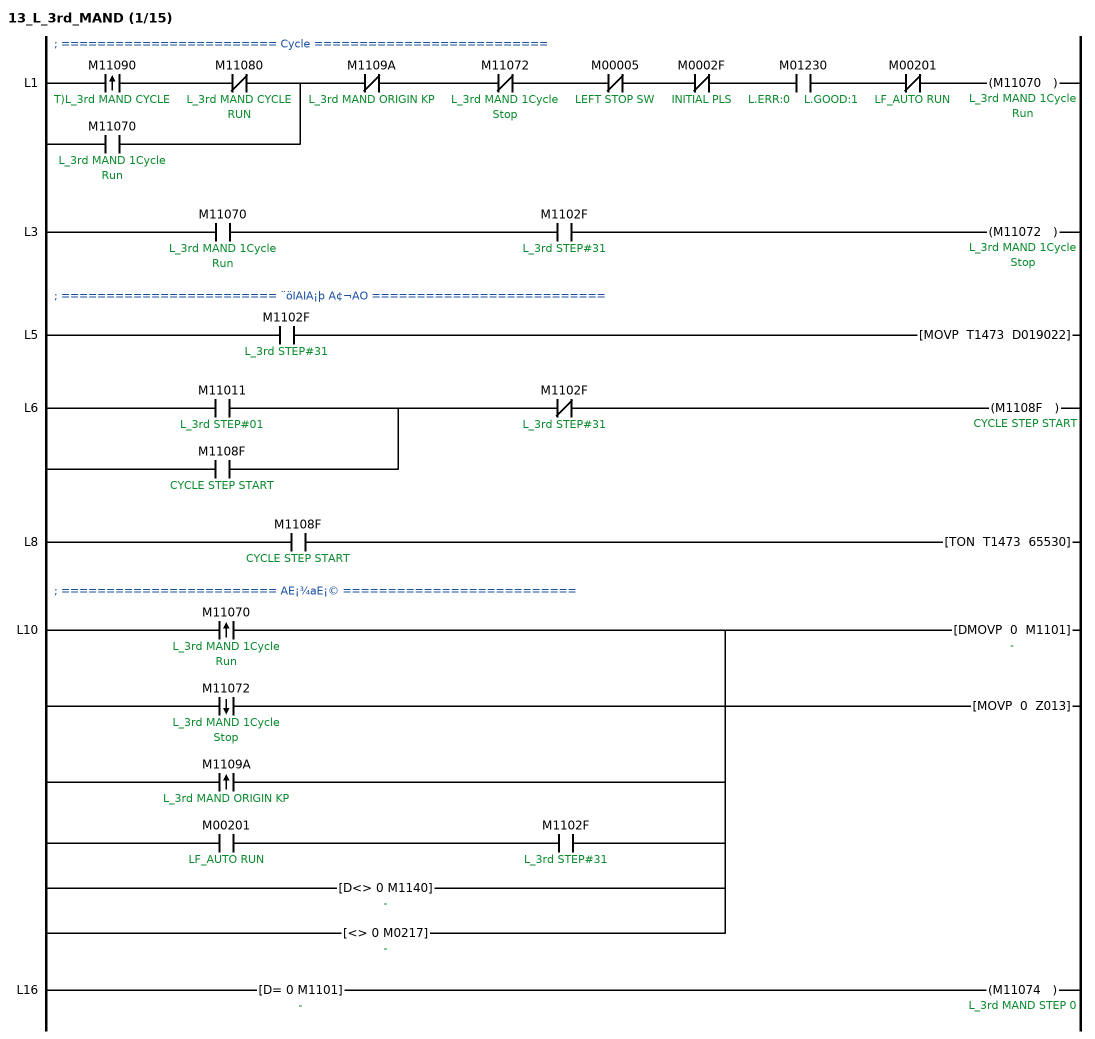
// ======================== Cycle ==========================
; L1
LOADP     M11090	// T)L_3rd MAND CYCLE
AND NOT   M11080	// L_3rd MAND CYCLE RUN
OR        M11070	// L_3rd MAND 1Cycle Run
AND NOT   M1109A	// L_3rd MAND ORIGIN KP
AND NOT   M11072	// L_3rd MAND 1Cycle Stop
AND NOT   M00005	// LEFT STOP SW
AND NOT   M0002F	// INITIAL PLS
AND       M01230	// L.ERR:0    L.GOOD:1
AND NOT   M00201	// LF_AUTO RUN
OUT       M11070	// L_3rd MAND 1Cycle Run
; L3
LOAD      M11070	// L_3rd MAND 1Cycle Run
AND       M1102F	// L_3rd STEP#31
OUT       M11072	// L_3rd MAND 1Cycle Stop
// ======================== ¨öIAIA¡þ A¢¬AO ==========================
; L5
LOAD      M1102F	// L_3rd STEP#31
MOVP      T1473 D019022
; L6
LOAD      M11011	// L_3rd STEP#01
OR        M1108F	// CYCLE STEP START
AND NOT   M1102F	// L_3rd STEP#31
OUT       M1108F	// CYCLE STEP START
; L8
LOAD      M1108F	// CYCLE STEP START
TON       T1473 65530
// ======================== AE¡¾aE¡© ==========================
; L10
LOADP     M11070	// L_3rd MAND 1Cycle Run
ORN       M11072	// L_3rd MAND 1Cycle Stop
ORP       M1109A	// L_3rd MAND ORIGIN KP
LOAD      M00201	// LF_AUTO RUN
AND       M1102F	// L_3rd STEP#31
OR LOAD
ORD<>     0 M1140	// -
OR<>      0 M0217	// -
DMOVP     0 M1101	// -
MOVP      0 Z013
; L16
LOADD=    0 M1101	// -
OUT       M11074	// L_3rd MAND STEP 0

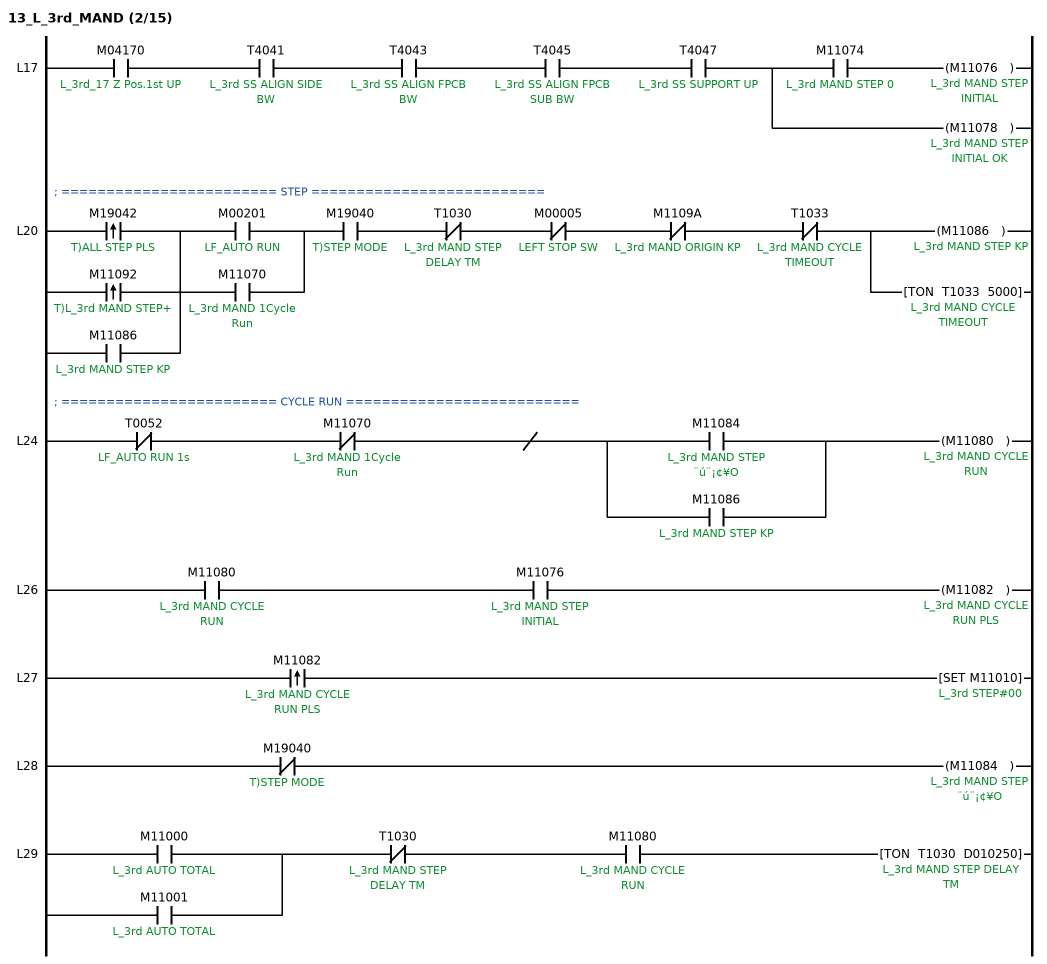
; L17
LOAD      M04170	// L_3rd_17 Z Pos.1st UP
AND       T4041	// L_3rd SS ALIGN SIDE BW
AND       T4043	// L_3rd SS ALIGN FPCB BW
AND       T4045	// L_3rd SS ALIGN FPCB SUB BW
AND       T4047	// L_3rd SS SUPPORT UP
MPUSH
AND       M11074	// L_3rd MAND STEP 0
OUT       M11076	// L_3rd MAND STEP INITIAL
MPOP
OUT       M11078	// L_3rd MAND STEP INITIAL OK
// ======================== STEP ==========================
; L20
LOADP     M19042	// T)ALL STEP PLS
ORP       M11092	// T)L_3rd MAND STEP+
OR        M11086	// L_3rd MAND STEP KP
LOAD      M00201	// LF_AUTO RUN
OR        M11070	// L_3rd MAND 1Cycle Run
AND LOAD
AND       M19040	// T)STEP MODE
AND NOT   T1030	// L_3rd MAND STEP DELAY TM
AND NOT   M00005	// LEFT STOP SW
AND NOT   M1109A	// L_3rd MAND ORIGIN KP
AND NOT   T1033	// L_3rd MAND CYCLE TIMEOUT
OUT       M11086	// L_3rd MAND STEP KP
TON       T1033 5000	// L_3rd MAND CYCLE TIMEOUT
// ======================== CYCLE RUN ==========================
; L24
LOAD NOT  T0052	// LF_AUTO RUN 1s
AND NOT   M11070	// L_3rd MAND 1Cycle Run
NOT
LOAD      M11084	// L_3rd MAND STEP ¨ú¨¡¢¥O
OR        M11086	// L_3rd MAND STEP KP
AND LOAD
OUT       M11080	// L_3rd MAND CYCLE RUN
; L26
LOAD      M11080	// L_3rd MAND CYCLE RUN
AND       M11076	// L_3rd MAND STEP INITIAL
OUT       M11082	// L_3rd MAND CYCLE RUN PLS
; L27
LOADP     M11082	// L_3rd MAND CYCLE RUN PLS
SET       M11010	// L_3rd STEP#00
; L28
LOAD NOT  M19040	// T)STEP MODE
OUT       M11084	// L_3rd MAND STEP ¨ú¨¡¢¥O
; L29
LOAD      M11000	// L_3rd AUTO TOTAL
OR        M11001	// L_3rd AUTO TOTAL
AND NOT   T1030	// L_3rd MAND STEP DELAY TM
AND       M11080	// L_3rd MAND CYCLE RUN
TON       T1030 D010250	// L_3rd MAND STEP DELAY TM

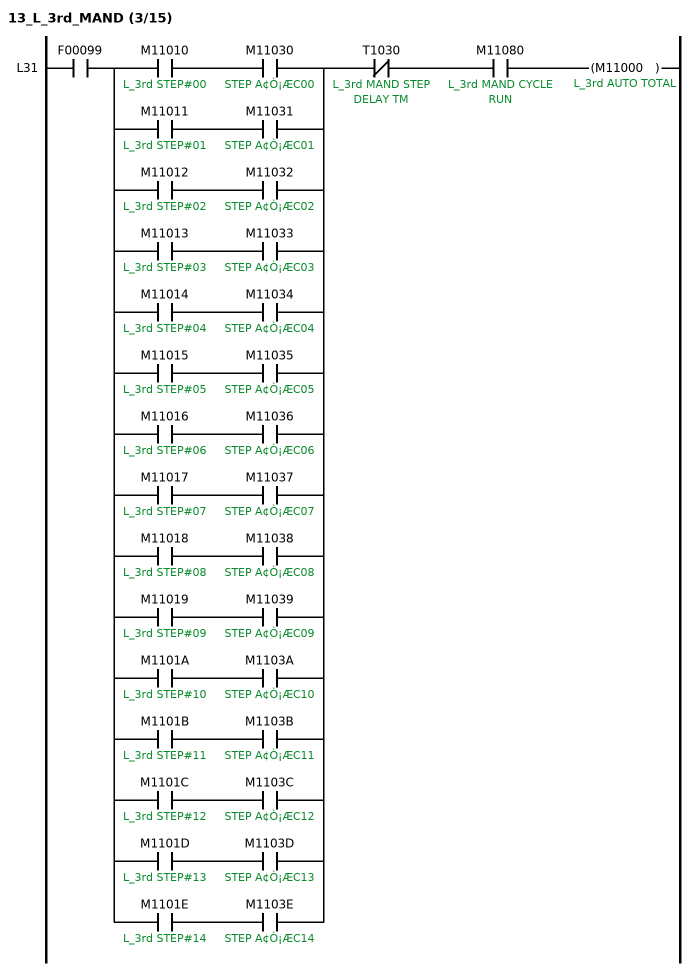
; L31
LOAD      F00099
LOAD      M11010	// L_3rd STEP#00
AND       M11030	// STEP A¢Ò¡ÆC00
LOAD      M11011	// L_3rd STEP#01
AND       M11031	// STEP A¢Ò¡ÆC01
OR LOAD
LOAD      M11012	// L_3rd STEP#02
AND       M11032	// STEP A¢Ò¡ÆC02
OR LOAD
LOAD      M11013	// L_3rd STEP#03
AND       M11033	// STEP A¢Ò¡ÆC03
OR LOAD
LOAD      M11014	// L_3rd STEP#04
AND       M11034	// STEP A¢Ò¡ÆC04
OR LOAD
LOAD      M11015	// L_3rd STEP#05
AND       M11035	// STEP A¢Ò¡ÆC05
OR LOAD
LOAD      M11016	// L_3rd STEP#06
AND       M11036	// STEP A¢Ò¡ÆC06
OR LOAD
LOAD      M11017	// L_3rd STEP#07
AND       M11037	// STEP A¢Ò¡ÆC07
OR LOAD
LOAD      M11018	// L_3rd STEP#08
AND       M11038	// STEP A¢Ò¡ÆC08
OR LOAD
LOAD      M11019	// L_3rd STEP#09
AND       M11039	// STEP A¢Ò¡ÆC09
OR LOAD
LOAD      M1101A	// L_3rd STEP#10
AND       M1103A	// STEP A¢Ò¡ÆC10
OR LOAD
LOAD      M1101B	// L_3rd STEP#11
AND       M1103B	// STEP A¢Ò¡ÆC11
OR LOAD
LOAD      M1101C	// L_3rd STEP#12
AND       M1103C	// STEP A¢Ò¡ÆC12
OR LOAD
LOAD      M1101D	// L_3rd STEP#13
AND       M1103D	// STEP A¢Ò¡ÆC13
OR LOAD
LOAD      M1101E	// L_3rd STEP#14
AND       M1103E	// STEP A¢Ò¡ÆC14
OR LOAD
AND LOAD
AND NOT   T1030	// L_3rd MAND STEP DELAY TM
AND       M11080	// L_3rd MAND CYCLE RUN
OUT       M11000	// L_3rd AUTO TOTAL

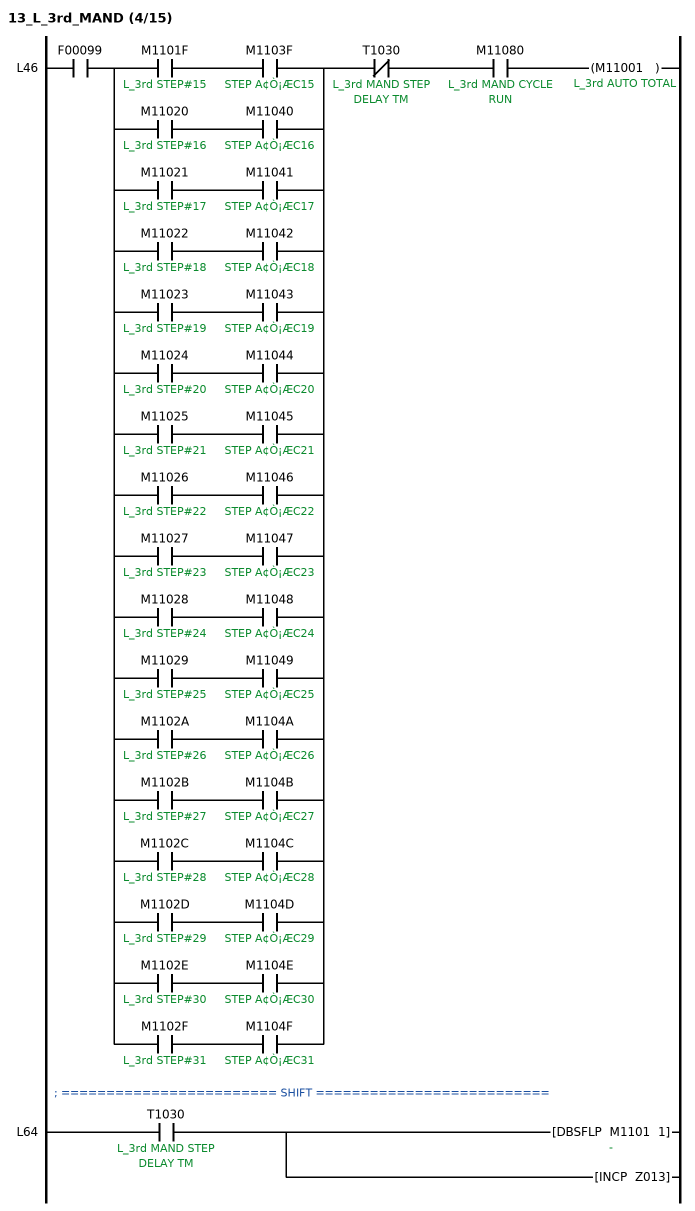
; L46
LOAD      F00099
LOAD      M1101F	// L_3rd STEP#15
AND       M1103F	// STEP A¢Ò¡ÆC15
LOAD      M11020	// L_3rd STEP#16
AND       M11040	// STEP A¢Ò¡ÆC16
OR LOAD
LOAD      M11021	// L_3rd STEP#17
AND       M11041	// STEP A¢Ò¡ÆC17
OR LOAD
LOAD      M11022	// L_3rd STEP#18
AND       M11042	// STEP A¢Ò¡ÆC18
OR LOAD
LOAD      M11023	// L_3rd STEP#19
AND       M11043	// STEP A¢Ò¡ÆC19
OR LOAD
LOAD      M11024	// L_3rd STEP#20
AND       M11044	// STEP A¢Ò¡ÆC20
OR LOAD
LOAD      M11025	// L_3rd STEP#21
AND       M11045	// STEP A¢Ò¡ÆC21
OR LOAD
LOAD      M11026	// L_3rd STEP#22
AND       M11046	// STEP A¢Ò¡ÆC22
OR LOAD
LOAD      M11027	// L_3rd STEP#23
AND       M11047	// STEP A¢Ò¡ÆC23
OR LOAD
LOAD      M11028	// L_3rd STEP#24
AND       M11048	// STEP A¢Ò¡ÆC24
OR LOAD
LOAD      M11029	// L_3rd STEP#25
AND       M11049	// STEP A¢Ò¡ÆC25
OR LOAD
LOAD      M1102A	// L_3rd STEP#26
AND       M1104A	// STEP A¢Ò¡ÆC26
OR LOAD
LOAD      M1102B	// L_3rd STEP#27
AND       M1104B	// STEP A¢Ò¡ÆC27
OR LOAD
LOAD      M1102C	// L_3rd STEP#28
AND       M1104C	// STEP A¢Ò¡ÆC28
OR LOAD
LOAD      M1102D	// L_3rd STEP#29
AND       M1104D	// STEP A¢Ò¡ÆC29
OR LOAD
LOAD      M1102E	// L_3rd STEP#30
AND       M1104E	// STEP A¢Ò¡ÆC30
OR LOAD
LOAD      M1102F	// L_3rd STEP#31
AND       M1104F	// STEP A¢Ò¡ÆC31
OR LOAD
AND LOAD
AND NOT   T1030	// L_3rd MAND STEP DELAY TM
AND       M11080	// L_3rd MAND CYCLE RUN
OUT       M11001	// L_3rd AUTO TOTAL
// ======================== SHIFT ==========================
; L64
LOAD      T1030	// L_3rd MAND STEP DELAY TM
DBSFLP    M1101 1	// -
INCP      Z013

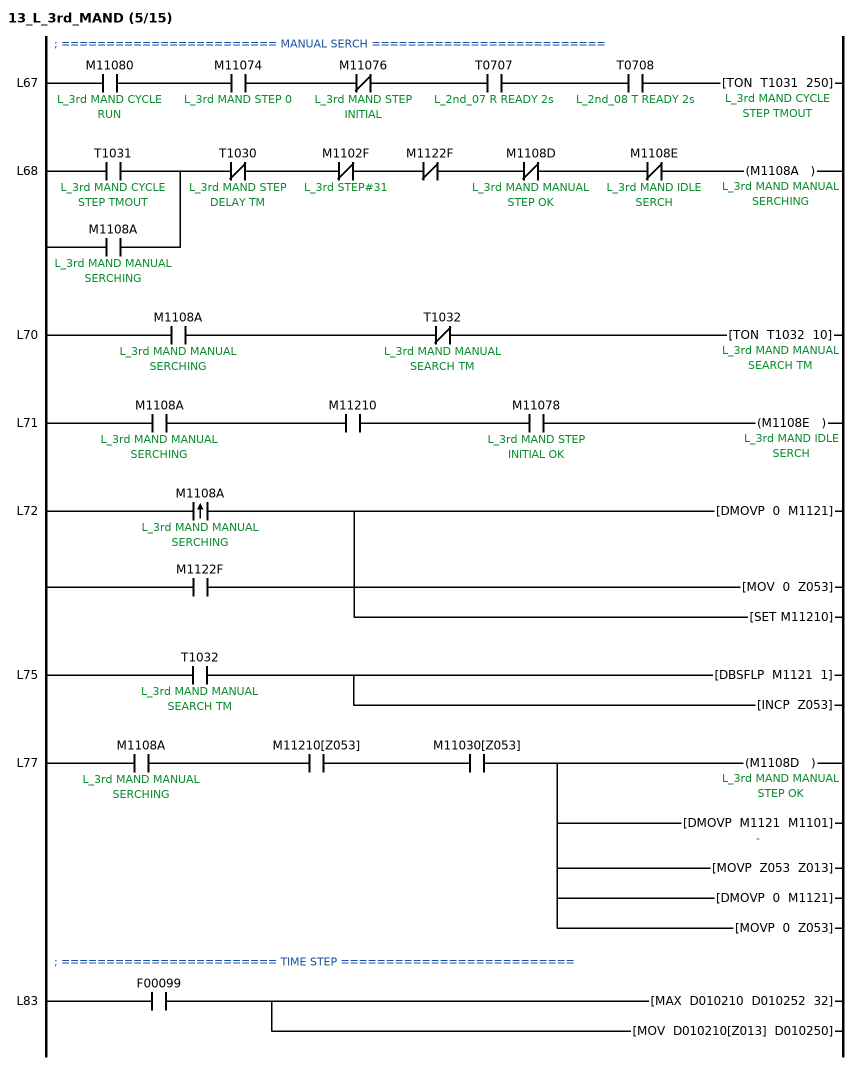
// ======================== MANUAL SERCH ==========================
; L67
LOAD      M11080	// L_3rd MAND CYCLE RUN
AND       M11074	// L_3rd MAND STEP 0
AND NOT   M11076	// L_3rd MAND STEP INITIAL
AND       T0707	// L_2nd_07 R READY 2s
AND       T0708	// L_2nd_08 T READY 2s
TON       T1031 250	// L_3rd MAND CYCLE STEP TMOUT
; L68
LOAD      T1031	// L_3rd MAND CYCLE STEP TMOUT
OR        M1108A	// L_3rd MAND MANUAL SERCHING
AND NOT   T1030	// L_3rd MAND STEP DELAY TM
AND NOT   M1102F	// L_3rd STEP#31
AND NOT   M1122F
AND NOT   M1108D	// L_3rd MAND MANUAL STEP OK
AND NOT   M1108E	// L_3rd MAND IDLE SERCH
OUT       M1108A	// L_3rd MAND MANUAL SERCHING
; L70
LOAD      M1108A	// L_3rd MAND MANUAL SERCHING
AND NOT   T1032	// L_3rd MAND MANUAL SEARCH TM
TON       T1032 10	// L_3rd MAND MANUAL SEARCH TM
; L71
LOAD      M1108A	// L_3rd MAND MANUAL SERCHING
AND       M11210
AND       M11078	// L_3rd MAND STEP INITIAL OK
OUT       M1108E	// L_3rd MAND IDLE SERCH
; L72
LOADP     M1108A	// L_3rd MAND MANUAL SERCHING
OR        M1122F
DMOVP     0 M1121
MOV       0 Z053
SET       M11210
; L75
LOAD      T1032	// L_3rd MAND MANUAL SEARCH TM
DBSFLP    M1121 1
INCP      Z053
; L77
LOAD      M1108A	// L_3rd MAND MANUAL SERCHING
AND       M11210[Z053]
AND       M11030[Z053]
OUT       M1108D	// L_3rd MAND MANUAL STEP OK
DMOVP     M1121 M1101	// -
MOVP      Z053 Z013
DMOVP     0 M1121
MOVP      0 Z053
// ======================== TIME STEP ==========================
; L83
LOAD      F00099
MAX       D010210 D010252 32
MOV       D010210[Z013] D010250

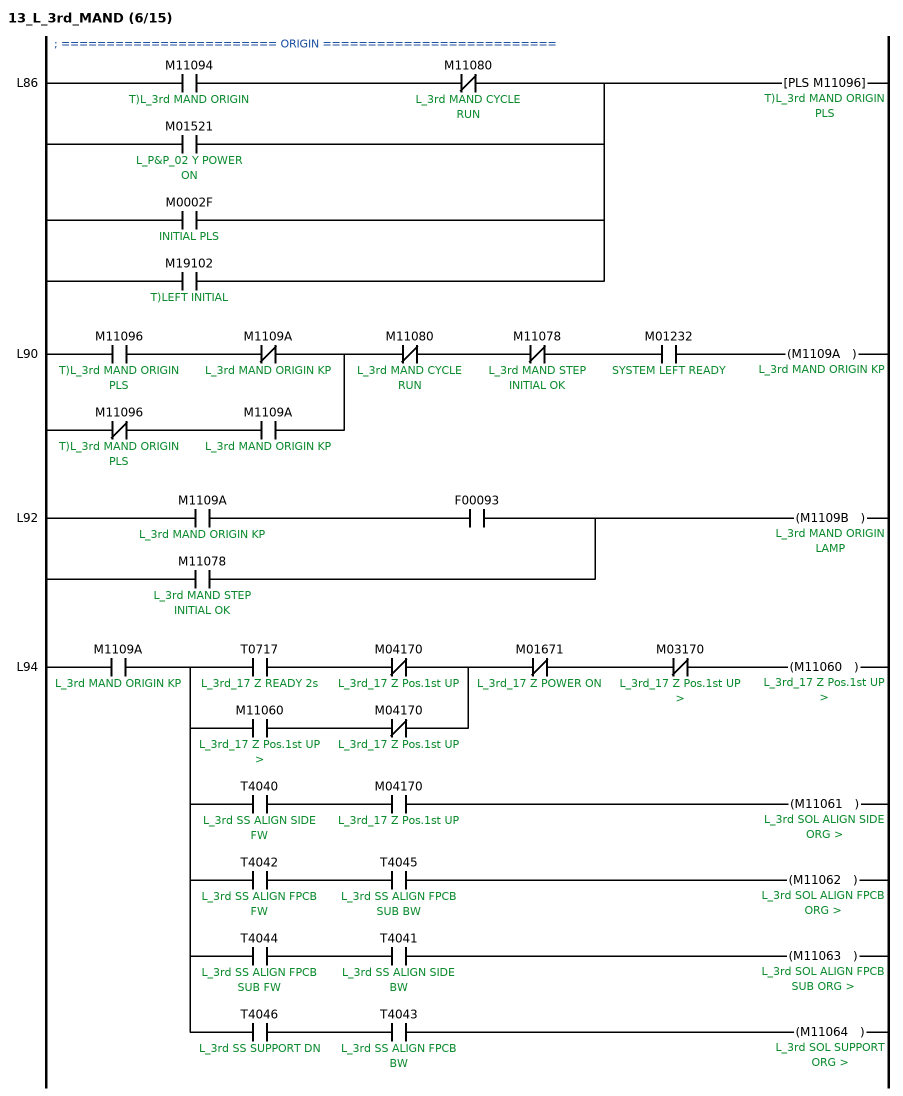
// ======================== ORIGIN ==========================
; L86
LOAD      M11094	// T)L_3rd MAND ORIGIN
AND NOT   M11080	// L_3rd MAND CYCLE RUN
OR        M01521	// L_P&P_02 Y POWER ON
OR        M0002F	// INITIAL PLS
OR        M19102	// T)LEFT INITIAL
OUTP      M11096	// T)L_3rd MAND ORIGIN PLS
; L90
LOAD      M11096	// T)L_3rd MAND ORIGIN PLS
AND NOT   M1109A	// L_3rd MAND ORIGIN KP
LOAD NOT  M11096	// T)L_3rd MAND ORIGIN PLS
AND       M1109A	// L_3rd MAND ORIGIN KP
OR LOAD
AND NOT   M11080	// L_3rd MAND CYCLE RUN
AND NOT   M11078	// L_3rd MAND STEP INITIAL OK
AND       M01232	// SYSTEM LEFT READY
OUT       M1109A	// L_3rd MAND ORIGIN KP
; L92
LOAD      M1109A	// L_3rd MAND ORIGIN KP
AND       F00093
OR        M11078	// L_3rd MAND STEP INITIAL OK
OUT       M1109B	// L_3rd MAND ORIGIN LAMP
; L94
LOAD      M1109A	// L_3rd MAND ORIGIN KP
MPUSH
LOAD      T0717	// L_3rd_17 Z READY 2s
AND NOT   M04170	// L_3rd_17 Z Pos.1st UP
LOAD      M11060	// L_3rd_17 Z Pos.1st UP >
AND NOT   M04170	// L_3rd_17 Z Pos.1st UP
OR LOAD
AND LOAD
AND NOT   M01671	// L_3rd_17 Z POWER ON
AND NOT   M03170	// L_3rd_17 Z Pos.1st UP >
OUT       M11060	// L_3rd_17 Z Pos.1st UP >
MLOAD
AND       T4040	// L_3rd SS ALIGN SIDE FW
AND       M04170	// L_3rd_17 Z Pos.1st UP
OUT       M11061	// L_3rd SOL ALIGN SIDE ORG >
MLOAD
AND       T4042	// L_3rd SS ALIGN FPCB FW
AND       T4045	// L_3rd SS ALIGN FPCB SUB BW
OUT       M11062	// L_3rd SOL ALIGN FPCB ORG >
MLOAD
AND       T4044	// L_3rd SS ALIGN FPCB SUB FW
AND       T4041	// L_3rd SS ALIGN SIDE BW
OUT       M11063	// L_3rd SOL ALIGN FPCB SUB ORG >
MPOP
AND       T4046	// L_3rd SS SUPPORT DN
AND       T4043	// L_3rd SS ALIGN FPCB BW
OUT       M11064	// L_3rd SOL SUPPORT ORG >

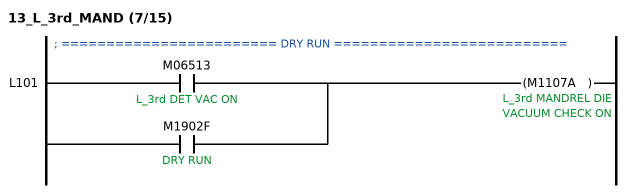
// ======================== DRY RUN ==========================
; L101
LOAD      M06513	// L_3rd DET VAC ON
OR        M1902F	// DRY RUN
OUT       M1107A	// L_3rd MANDREL DIE VACUUM CHECK ON

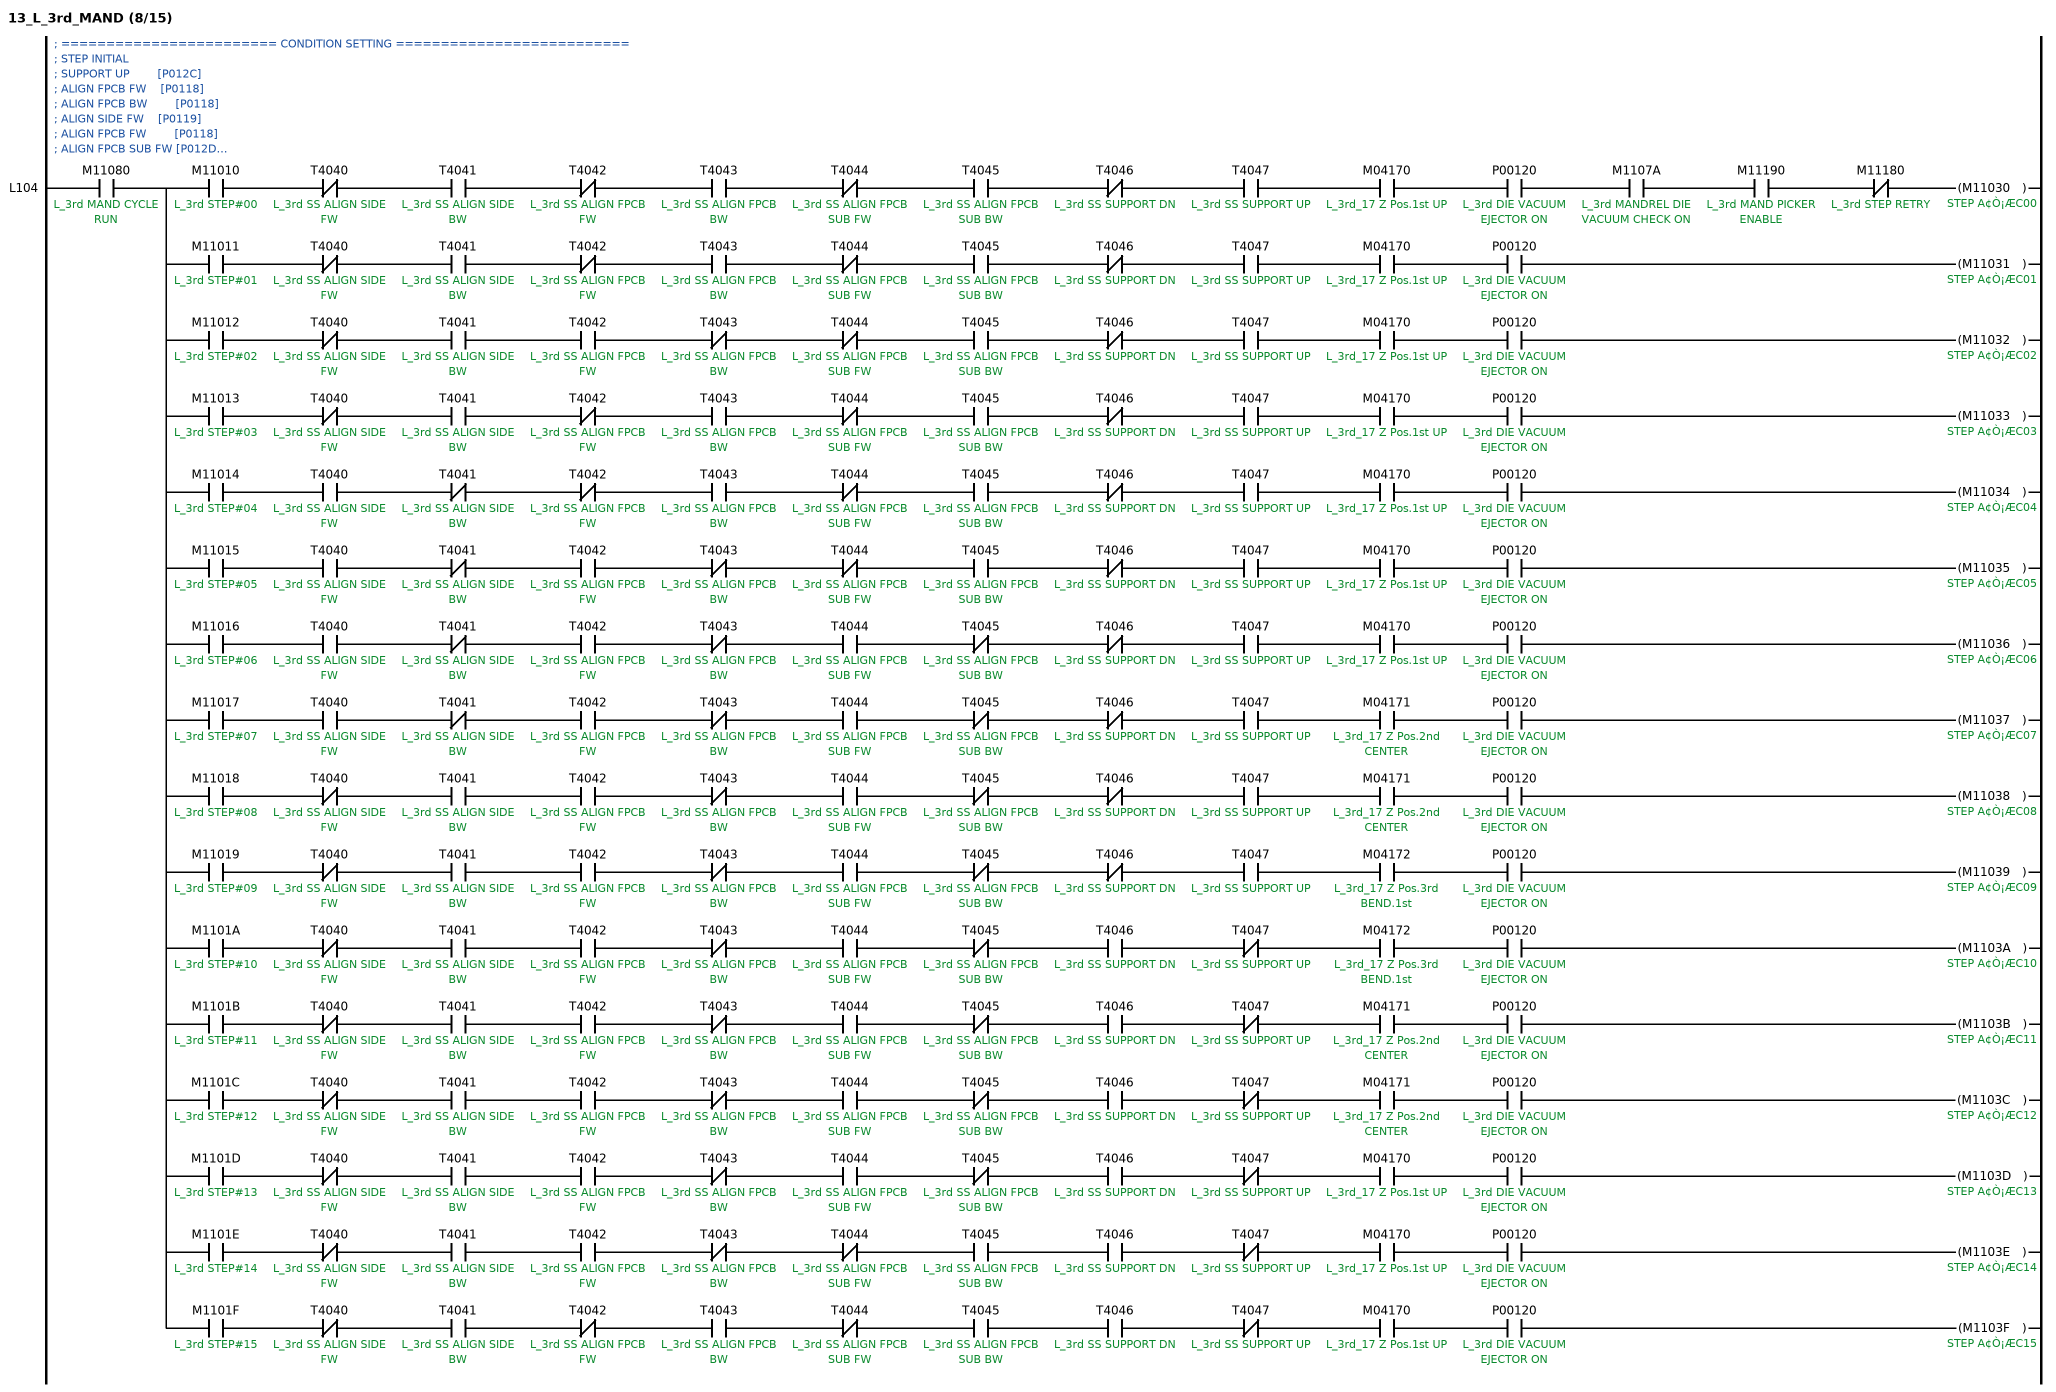
// ======================== CONDITION SETTING ==========================
; L104
LOAD      M11080	// L_3rd MAND CYCLE RUN
MPUSH
AND       M11010	// L_3rd STEP#00
AND NOT   T4040	// L_3rd SS ALIGN SIDE FW
AND       T4041	// L_3rd SS ALIGN SIDE BW
AND NOT   T4042	// L_3rd SS ALIGN FPCB FW
AND       T4043	// L_3rd SS ALIGN FPCB BW
AND NOT   T4044	// L_3rd SS ALIGN FPCB SUB FW
AND       T4045	// L_3rd SS ALIGN FPCB SUB BW
AND NOT   T4046	// L_3rd SS SUPPORT DN
AND       T4047	// L_3rd SS SUPPORT UP
AND       M04170	// L_3rd_17 Z Pos.1st UP
AND       P00120	// L_3rd DIE VACUUM EJECTOR ON
AND       M1107A	// L_3rd MANDREL DIE VACUUM CHECK ON
AND       M11190	// L_3rd MAND PICKER ENABLE
AND NOT   M11180	// L_3rd STEP RETRY
OUT       M11030	// STEP A¢Ò¡ÆC00
MLOAD
AND       M11011	// L_3rd STEP#01
AND NOT   T4040	// L_3rd SS ALIGN SIDE FW
AND       T4041	// L_3rd SS ALIGN SIDE BW
AND NOT   T4042	// L_3rd SS ALIGN FPCB FW
AND       T4043	// L_3rd SS ALIGN FPCB BW
AND NOT   T4044	// L_3rd SS ALIGN FPCB SUB FW
AND       T4045	// L_3rd SS ALIGN FPCB SUB BW
AND NOT   T4046	// L_3rd SS SUPPORT DN
AND       T4047	// L_3rd SS SUPPORT UP
AND       M04170	// L_3rd_17 Z Pos.1st UP
AND       P00120	// L_3rd DIE VACUUM EJECTOR ON
OUT       M11031	// STEP A¢Ò¡ÆC01
MLOAD
AND       M11012	// L_3rd STEP#02
AND NOT   T4040	// L_3rd SS ALIGN SIDE FW
AND       T4041	// L_3rd SS ALIGN SIDE BW
AND       T4042	// L_3rd SS ALIGN FPCB FW
AND NOT   T4043	// L_3rd SS ALIGN FPCB BW
AND NOT   T4044	// L_3rd SS ALIGN FPCB SUB FW
AND       T4045	// L_3rd SS ALIGN FPCB SUB BW
AND NOT   T4046	// L_3rd SS SUPPORT DN
AND       T4047	// L_3rd SS SUPPORT UP
AND       M04170	// L_3rd_17 Z Pos.1st UP
AND       P00120	// L_3rd DIE VACUUM EJECTOR ON
OUT       M11032	// STEP A¢Ò¡ÆC02
MLOAD
AND       M11013	// L_3rd STEP#03
AND NOT   T4040	// L_3rd SS ALIGN SIDE FW
AND       T4041	// L_3rd SS ALIGN SIDE BW
AND NOT   T4042	// L_3rd SS ALIGN FPCB FW
AND       T4043	// L_3rd SS ALIGN FPCB BW
AND NOT   T4044	// L_3rd SS ALIGN FPCB SUB FW
AND       T4045	// L_3rd SS ALIGN FPCB SUB BW
AND NOT   T4046	// L_3rd SS SUPPORT DN
AND       T4047	// L_3rd SS SUPPORT UP
AND       M04170	// L_3rd_17 Z Pos.1st UP
AND       P00120	// L_3rd DIE VACUUM EJECTOR ON
OUT       M11033	// STEP A¢Ò¡ÆC03
MLOAD
AND       M11014	// L_3rd STEP#04
AND       T4040	// L_3rd SS ALIGN SIDE FW
AND NOT   T4041	// L_3rd SS ALIGN SIDE BW
AND NOT   T4042	// L_3rd SS ALIGN FPCB FW
AND       T4043	// L_3rd SS ALIGN FPCB BW
AND NOT   T4044	// L_3rd SS ALIGN FPCB SUB FW
AND       T4045	// L_3rd SS ALIGN FPCB SUB BW
AND NOT   T4046	// L_3rd SS SUPPORT DN
AND       T4047	// L_3rd SS SUPPORT UP
AND       M04170	// L_3rd_17 Z Pos.1st UP
AND       P00120	// L_3rd DIE VACUUM EJECTOR ON
OUT       M11034	// STEP A¢Ò¡ÆC04
MLOAD
AND       M11015	// L_3rd STEP#05
AND       T4040	// L_3rd SS ALIGN SIDE FW
AND NOT   T4041	// L_3rd SS ALIGN SIDE BW
AND       T4042	// L_3rd SS ALIGN FPCB FW
AND NOT   T4043	// L_3rd SS ALIGN FPCB BW
AND NOT   T4044	// L_3rd SS ALIGN FPCB SUB FW
AND       T4045	// L_3rd SS ALIGN FPCB SUB BW
AND NOT   T4046	// L_3rd SS SUPPORT DN
AND       T4047	// L_3rd SS SUPPORT UP
AND       M04170	// L_3rd_17 Z Pos.1st UP
AND       P00120	// L_3rd DIE VACUUM EJECTOR ON
OUT       M11035	// STEP A¢Ò¡ÆC05
MLOAD
AND       M11016	// L_3rd STEP#06
AND       T4040	// L_3rd SS ALIGN SIDE FW
AND NOT   T4041	// L_3rd SS ALIGN SIDE BW
AND       T4042	// L_3rd SS ALIGN FPCB FW
AND NOT   T4043	// L_3rd SS ALIGN FPCB BW
AND       T4044	// L_3rd SS ALIGN FPCB SUB FW
AND NOT   T4045	// L_3rd SS ALIGN FPCB SUB BW
AND NOT   T4046	// L_3rd SS SUPPORT DN
AND       T4047	// L_3rd SS SUPPORT UP
AND       M04170	// L_3rd_17 Z Pos.1st UP
AND       P00120	// L_3rd DIE VACUUM EJECTOR ON
OUT       M11036	// STEP A¢Ò¡ÆC06
MLOAD
AND       M11017	// L_3rd STEP#07
AND       T4040	// L_3rd SS ALIGN SIDE FW
AND NOT   T4041	// L_3rd SS ALIGN SIDE BW
AND       T4042	// L_3rd SS ALIGN FPCB FW
AND NOT   T4043	// L_3rd SS ALIGN FPCB BW
AND       T4044	// L_3rd SS ALIGN FPCB SUB FW
AND NOT   T4045	// L_3rd SS ALIGN FPCB SUB BW
AND NOT   T4046	// L_3rd SS SUPPORT DN
AND       T4047	// L_3rd SS SUPPORT UP
AND       M04171	// L_3rd_17 Z Pos.2nd CENTER
AND       P00120	// L_3rd DIE VACUUM EJECTOR ON
OUT       M11037	// STEP A¢Ò¡ÆC07
MLOAD
AND       M11018	// L_3rd STEP#08
AND NOT   T4040	// L_3rd SS ALIGN SIDE FW
AND       T4041	// L_3rd SS ALIGN SIDE BW
AND       T4042	// L_3rd SS ALIGN FPCB FW
AND NOT   T4043	// L_3rd SS ALIGN FPCB BW
AND       T4044	// L_3rd SS ALIGN FPCB SUB FW
AND NOT   T4045	// L_3rd SS ALIGN FPCB SUB BW
AND NOT   T4046	// L_3rd SS SUPPORT DN
AND       T4047	// L_3rd SS SUPPORT UP
AND       M04171	// L_3rd_17 Z Pos.2nd CENTER
AND       P00120	// L_3rd DIE VACUUM EJECTOR ON
OUT       M11038	// STEP A¢Ò¡ÆC08
MLOAD
AND       M11019	// L_3rd STEP#09
AND NOT   T4040	// L_3rd SS ALIGN SIDE FW
AND       T4041	// L_3rd SS ALIGN SIDE BW
AND       T4042	// L_3rd SS ALIGN FPCB FW
AND NOT   T4043	// L_3rd SS ALIGN FPCB BW
AND       T4044	// L_3rd SS ALIGN FPCB SUB FW
AND NOT   T4045	// L_3rd SS ALIGN FPCB SUB BW
AND NOT   T4046	// L_3rd SS SUPPORT DN
AND       T4047	// L_3rd SS SUPPORT UP
AND       M04172	// L_3rd_17 Z Pos.3rd BEND.1st
AND       P00120	// L_3rd DIE VACUUM EJECTOR ON
OUT       M11039	// STEP A¢Ò¡ÆC09
MLOAD
AND       M1101A	// L_3rd STEP#10
AND NOT   T4040	// L_3rd SS ALIGN SIDE FW
AND       T4041	// L_3rd SS ALIGN SIDE BW
AND       T4042	// L_3rd SS ALIGN FPCB FW
AND NOT   T4043	// L_3rd SS ALIGN FPCB BW
AND       T4044	// L_3rd SS ALIGN FPCB SUB FW
AND NOT   T4045	// L_3rd SS ALIGN FPCB SUB BW
AND       T4046	// L_3rd SS SUPPORT DN
AND NOT   T4047	// L_3rd SS SUPPORT UP
AND       M04172	// L_3rd_17 Z Pos.3rd BEND.1st
AND       P00120	// L_3rd DIE VACUUM EJECTOR ON
OUT       M1103A	// STEP A¢Ò¡ÆC10
MLOAD
AND       M1101B	// L_3rd STEP#11
AND NOT   T4040	// L_3rd SS ALIGN SIDE FW
AND       T4041	// L_3rd SS ALIGN SIDE BW
AND       T4042	// L_3rd SS ALIGN FPCB FW
AND NOT   T4043	// L_3rd SS ALIGN FPCB BW
AND       T4044	// L_3rd SS ALIGN FPCB SUB FW
AND NOT   T4045	// L_3rd SS ALIGN FPCB SUB BW
AND       T4046	// L_3rd SS SUPPORT DN
AND NOT   T4047	// L_3rd SS SUPPORT UP
AND       M04171	// L_3rd_17 Z Pos.2nd CENTER
AND       P00120	// L_3rd DIE VACUUM EJECTOR ON
OUT       M1103B	// STEP A¢Ò¡ÆC11
MLOAD
AND       M1101C	// L_3rd STEP#12
AND NOT   T4040	// L_3rd SS ALIGN SIDE FW
AND       T4041	// L_3rd SS ALIGN SIDE BW
AND       T4042	// L_3rd SS ALIGN FPCB FW
AND NOT   T4043	// L_3rd SS ALIGN FPCB BW
AND       T4044	// L_3rd SS ALIGN FPCB SUB FW
AND NOT   T4045	// L_3rd SS ALIGN FPCB SUB BW
AND       T4046	// L_3rd SS SUPPORT DN
AND NOT   T4047	// L_3rd SS SUPPORT UP
AND       M04171	// L_3rd_17 Z Pos.2nd CENTER
AND       P00120	// L_3rd DIE VACUUM EJECTOR ON
OUT       M1103C	// STEP A¢Ò¡ÆC12
MLOAD
AND       M1101D	// L_3rd STEP#13
AND NOT   T4040	// L_3rd SS ALIGN SIDE FW
AND       T4041	// L_3rd SS ALIGN SIDE BW
AND       T4042	// L_3rd SS ALIGN FPCB FW
AND NOT   T4043	// L_3rd SS ALIGN FPCB BW
AND       T4044	// L_3rd SS ALIGN FPCB SUB FW
AND NOT   T4045	// L_3rd SS ALIGN FPCB SUB BW
AND       T4046	// L_3rd SS SUPPORT DN
AND NOT   T4047	// L_3rd SS SUPPORT UP
AND       M04170	// L_3rd_17 Z Pos.1st UP
AND       P00120	// L_3rd DIE VACUUM EJECTOR ON
OUT       M1103D	// STEP A¢Ò¡ÆC13
MLOAD
AND       M1101E	// L_3rd STEP#14
AND NOT   T4040	// L_3rd SS ALIGN SIDE FW
AND       T4041	// L_3rd SS ALIGN SIDE BW
AND       T4042	// L_3rd SS ALIGN FPCB FW
AND NOT   T4043	// L_3rd SS ALIGN FPCB BW
AND NOT   T4044	// L_3rd SS ALIGN FPCB SUB FW
AND       T4045	// L_3rd SS ALIGN FPCB SUB BW
AND       T4046	// L_3rd SS SUPPORT DN
AND NOT   T4047	// L_3rd SS SUPPORT UP
AND       M04170	// L_3rd_17 Z Pos.1st UP
AND       P00120	// L_3rd DIE VACUUM EJECTOR ON
OUT       M1103E	// STEP A¢Ò¡ÆC14
MPOP
AND       M1101F	// L_3rd STEP#15
AND NOT   T4040	// L_3rd SS ALIGN SIDE FW
AND       T4041	// L_3rd SS ALIGN SIDE BW
AND NOT   T4042	// L_3rd SS ALIGN FPCB FW
AND       T4043	// L_3rd SS ALIGN FPCB BW
AND NOT   T4044	// L_3rd SS ALIGN FPCB SUB FW
AND       T4045	// L_3rd SS ALIGN FPCB SUB BW
AND       T4046	// L_3rd SS SUPPORT DN
AND NOT   T4047	// L_3rd SS SUPPORT UP
AND       M04170	// L_3rd_17 Z Pos.1st UP
AND       P00120	// L_3rd DIE VACUUM EJECTOR ON
OUT       M1103F	// STEP A¢Ò¡ÆC15
// output comment: STEP INITIAL
// output comment: SUPPORT UP        [P012C]
// output comment: ALIGN FPCB FW    [P0118]
// output comment: ALIGN FPCB BW        [P0118]
// output comment: ALIGN SIDE FW    [P0119]
// output comment: ALIGN FPCB FW        [P0118]
// output comment: ALIGN FPCB SUB FW [P012D]
// output comment: L_3rd_17 Z Pos.2nd CENTER >
// output comment: ALIGN SIDE BW      [P0119]
// output comment: L_3rd_17 Z Pos.3rd BEND.1st >
// output comment: SUPPORT DN      [P012C]
// output comment: L_3rd_17 Z Pos.2nd CENTER >
// output comment: L_3rd_17 Z Pos.1st      UP >
// output comment: ALIGN FPCB SUB BW [P012D]
// output comment: ALIGN FPCB BW    [P0118]

